	nCurrentPhotonEnergyBitmask : UINT;
	nTargetPhotonEnergyBitmask : UINT;
END_VAR

// Update PVs
fbHgvpuElectronEnergy();

fElectronEnergyVal := fbHgvpuElectronEnergy.fValue;
bElectronEnergyValid := fbHgvpuElectronEnergy.bValid;

fbHgvpu(fbElectronEnergy:=fbHgvpuElectronEnergy);

//Update BP
nCurrentPhotonEnergyBitmask := F_eVRangeCalculator(fbHgvpu.fCurrentPhotonEnergy, nCurrentPhotonEnergyBitmask);
nTargetPhotonEnergyBitmask := F_eVRangeCalculator(fbHgvpu.fTargetPhotonEnergy, nTargetPhotonEnergyBitmask);

BP.neVRange := nCurrentPhotonEnergyBitmask OR nTargetPhotonEnergyBitmask;

END_FUNCTION_BLOCK

// MajorComponents/PMPS_MPS_Interface/FB_BeamClassOutputs
(*
Sets the beam class assertion lines for a given beam class.
*)
FUNCTION_BLOCK FB_BeamClassOutputs
VAR_INPUT
    BP : ST_BeamParams;
END_VAR
VAR_OUTPUT
END_VAR
VAR
    nBeamClass   :    BYTE;
    wBeamClass    :    BYTE;

    InitCounter: BYTE;
    counter    :    INT;
    
    // Beam class lines are restricted to 8 channels in the current design, since
    // there are no plans to use all 16. Channels 1-7 may be allocated to any other
    // beam classes so long as they are ordered least to greatest.
    // Channel 8 is reserved for full beam.
    {attribute 'pytmc' := 'pv: BeamClassChannel
        io: i
        field: DESC Hardwire channel state'}
        epicsBitmap : WORD;
        
    {attribute 'TcLinkTo' := '[1] := TIIB[PMPS_Premp]^Channel 1^Output;
                              [2] := TIIB[PMPS_Premp]^Channel 2^Output;
                              [3] := TIIB[PMPS_Premp]^Channel 3^Output;
                              [4] := TIIB[PMPS_Premp]^Channel 4^Output;
                              
                              [5] := TIIB[PMPS_Premp]^Channel 5^Output;
                              [6] := TIIB[PMPS_Premp]^Channel 6^Output;
                              [7] := TIIB[PMPS_Premp]^Channel 7^Output;
                              [8] := TIIB[PMPS_Premp]^Channel 8^Output;'} // 8 - Full beam
    q_BC_ASSERTION_LINES    AT    %Q*    : ARRAY [1..MAX_BEAM_CLASS_LINES] OF    BOOL;
END_VAR
VAR CONSTANT
    MAX_BEAM_CLASS_LINES : BYTE := 8;
    BC_1HZ : BYTE := 1;
    BC_10HZ : BYTE := 2;
    BC_FULL : BYTE := 16;
END_VAR


// Determine BC
IF BP.nRate >= 120 THEN
    nBeamClass := BC_FULL;
ELSIF BP.nRate >= 10 THEN
    nBeamClass := BC_10HZ;
ELSIF BP.nRate >= 1 THEN
    nBeamClass := BC_1HZ;
ELSE
	nBeamClass := 0;
END_IF


//Assert Beam Class
////////////////////////////////////
//0x0 = 0000 0000 0000 0000
//0x1 = 0000 0000 0000 0001
//0xF = 1111 1111 1111 1111

//Initialize BC lines to zero on every pass
FOR InitCounter := 1 TO MAX_BEAM_CLASS_LINES DO
    q_BC_ASSERTION_LINES[InitCounter] := FALSE;
END_FOR

//Set BC lines according to beam class
//A BC of 0x0 would pass over this loop, setting none of the lines high
// , as FOR loops check the initialized variable at the top to see if it's >
// than the "TO" variable.
FOR wBeamClass:=1 TO MIN(MAX_BEAM_CLASS_LINES-1, nBeamClass) DO
    q_BC_ASSERTION_LINES[wBeamClass] := TRUE;
END_FOR

q_BC_ASSERTION_LINES[8] := nBeamClass = 16; //Set channel 8 true if BC is 16


// Readbacks for EPICS
epicsBitmap.0 := q_BC_ASSERTION_LINES[1];
epicsBitmap.1 := q_BC_ASSERTION_LINES[2];
epicsBitmap.2 := q_BC_ASSERTION_LINES[3];
epicsBitmap.3 := q_BC_ASSERTION_LINES[4];

epicsBitmap.4 := q_BC_ASSERTION_LINES[5];
epicsBitmap.5 := q_BC_ASSERTION_LINES[6];
epicsBitmap.6 := q_BC_ASSERTION_LINES[7];
epicsBitmap.7 := q_BC_ASSERTION_LINES[8];

END_FUNCTION_BLOCK

// MajorComponents/PMPS_MPS_Interface/FB_CTLS_Outputs
(*
Controls auxiliary beam class outputs.

1-3 are mapped to control the Cu beamline rate via the LCLS II MPS.

Maps beam rate requests to 1, 10, or full rate beam for Cu linac.

*)
FUNCTION_BLOCK FB_CTLS_Outputs
VAR_INPUT
    BP    :    ST_BeamParams;
END_VAR
VAR_OUTPUT
END_VAR
VAR
    {attribute 'pytmc' := 'pv: CTLSChannel
        io: i
        field: DESC CTLS Rate Control hardwire channel state'}
    epicsBitmap : WORD;
        
    {attribute 'TcLinkTo' := '[1] := TIIB[PMPS_Premp]^Channel 9^Output;
                              [2] := TIIB[PMPS_Premp]^Channel 10^Output;
                              [3] := TIIB[PMPS_Premp]^Channel 11^Output;'}
    q_CLTS_ASSERTION_LINES    AT    %Q*    : ARRAY [1..3] OF    BOOL;  
    
    
    
END_VAR


// CLTS 1Hz
q_CLTS_ASSERTION_LINES[1] := BP.nRate >= 1;
// CLTS 10Hz
q_CLTS_ASSERTION_LINES[2] := BP.nRate >= 10;
// CLTS Full rate
q_CLTS_ASSERTION_LINES[3] := BP.nRate >= 120;


epicsBitMap.0 := q_CLTS_ASSERTION_LINES[1];
epicsBitMap.1 := q_CLTS_ASSERTION_LINES[2];
epicsBitMap.2 := q_CLTS_ASSERTION_LINES[3];

END_FUNCTION_BLOCK

// MajorComponents/PMPS_MPS_Interface/FB_PhotonEnergyWatcher
(*
A. Wallace 2019-4-22
The photon energy watcher ensures the current and target photon energy is within
the arbirated bounds. Target in this case means, the calculated target photon energy
from the PVs that control the mechatronics of the undulators/ the electron energy.

If there are control PVs that match the monitor PVs, the control PVs are used to 
calculate a "target" photon energy. This is supposed to cover when the undulators/
electron energy is transitioning.

The abritrated bounds come from a simple AND of all the permitted ranges. See
the arbitrate action of the arbiter FB.

Note, this protection logic does not account for beam-off when determining fast-fault
status. If a device is requesting a limited range of eV, this request must be honored,
regardless of current beam-rate.
*)
{attribute 'reflection'}
FUNCTION_BLOCK FB_PhotonEnergyWatcher
VAR_INPUT
    i_stCurrentBeamParams    :    ST_BeamParams; //Link to global beam params
    i_stMachineTargetBeamParams    :    ST_BeamParams; //Link to global machine target beam params
    i_stRequestedBeamParams    :    ST_BeamParams; //Link to arbiter output or beam param. requestor
    // Reset fault
    i_xReset: BOOL;
    sName : STRING := 'PhotonEnergyWatcher';
END_VAR
VAR_OUTPUT
END_VAR
VAR_IN_OUT
    io_fbFFHWO    :    FB_HardwareFFOutput;
END_VAR
VAR
    xPhotonEnergyWithinBounds    :    BOOL;
    fbFF    :    FB_FastFault :=(
        i_DevName := sName,
        i_Desc := 'Fault occurs when the calculated machine photon energy (K value calculated by undulator gap, and electron energy) falls outside the permitted range.',
        i_TypeCode := 7 );
        
   {attribute 'pytmc' := '
        pv: ResidualPhotonEnergies
		io: i
        archive: 1Hz monitor
        field: DESC Portions of beam eV not permitted
        field: EGU eV-bitmask
    '}
    evResidual : WORD;
    
    fbLog : FB_LogMessage := (
        eSubSystem := E_Subsystem.MPS,
        eSevr := TcEventSeverity.Critical
        );
    bLogOneShot : BOOL;
    sDevName : T_MaxString := 'Photon Energy Watcher';
    
    fbGetHN : FB_GetHostName;
    bInit : BOOL := TRUE;
    
    {attribute 'instance-path'}
    {attribute 'noinit'}
    sPath    :    T_MaxString;
    
    fbStr : FB_FormatString := (
        sOut := 'Non-zero photon energy residual: %16b; Req: %16b; Act: %16b');
END_VAR

IF bInit THEN
    fbGetHN(bExecute:=TRUE);
    bInit R= NOT fbGetHN.bBusy;
END_IF
    
xPhotonEnergyWithinBounds := (i_stCurrentBeamParams.neVRange AND i_stRequestedBeamParams.neVRange) = i_stCurrentBeamParams.neVRange;

evResidual := (i_stCurrentBeamParams.neVRange XOR i_stRequestedBeamParams.neVRange) AND i_stCurrentBeamParams.neVRange;

IF evResidual <> 0 AND bLogOneShot THEN
    fbLog.sJson := F_PMPS_JSON(
        CONCAT(fbGetHN.sHostName, sDevName),
        sPath,
        PMPS_CODES.PEW_FAULT);
    
    fbStr.arg1 := F_WORD(evResidual);
    fbStr.arg2 := F_WORD(i_stCurrentBeamParams.neVRange);
    fbStr.arg3 := F_WORD(i_stRequestedBeamParams.neVRange);
    
    fbStr();
        
    fbLog(sMsg:=fbStr.sOut);
    bLogOneShot := FALSE;
ELSIF evResidual = 0 THEN
    bLogOneShot := TRUE;
END_IF

fbFF(i_xOK := xPhotonEnergyWithinBounds,
    io_fbFFHWO := io_fbFFHWO,);

END_FUNCTION_BLOCK

// MajorComponents/SimulationFB/FB_eVSimulator
(* eV Simulator
A. Wallace 2019-8-30

Adds noise to the eV and changes eV position occasionally.
*)
FUNCTION_BLOCK FB_eVSimulator
VAR_INPUT
    NoiseLevel	:	REAL	:= 0; // eV Noise
    ChangeTime : TIME := T#10S;
END_VAR
VAR_OUTPUT
    eV	:	REAL := 300;
END_VAR
VAR
    eVRange : REAL := 1600;
    timer: TON;
    eVRand	:	DRAND :=(Seed:=0);
    NoiseRand : DRAND := (Seed:=0);
END_VAR


timer(in:=TRUE, PT:=ChangeTime);

//Occasionally change eV
IF timer.Q THEN
    timer(in:=FALSE);
    eVRand();
    eV := LIMIT(0, eVRange*LREAL_TO_REAL(eVRand.Num), eVRange);
END_IF

// Noise generation
NoiseRand();
eV := eV + NoiseLevel*LREAL_TO_REAL(NoiseRand.Num);
NoiseRand();
eV := LIMIT(0, ev - NoiseLevel*LREAL_TO_REAL(NoiseRand.Num), eVRange);

END_FUNCTION_BLOCK

// MajorComponents/SimulationFB/FB_MachineSimulator
(* Simulates the machine responding to requests by adding a bit of delay/ ramps
*)
FUNCTION_BLOCK FB_MachineSimulator
VAR_INPUT
    i_stAssertedParams    :    ST_BeamParams;
    i_xFault    :    BOOL;
    
    xEnableAtt : BOOL;
    xEnablePE : BOOL;
    xEnableRate : BOOL;
END_VAR
VAR_IN_OUT
    iq_stMachineParams    :    ST_BeamParams;
END_VAR
VAR
    nTargetTran: UINT;
    tonTranTimer    :    TON := (
        PT := T#2S
        );
    fTargetPP_mJ: REAL;
    tonPPETimer: TON := (
        PT := T#2S
    );
END_VAR


//Attenuation
IF xEnableAtt THEN
    IF i_stAssertedParams.nTran <> nTargetTran THEN
        tonTranTimer(IN:=FALSE);
        nTargetTran := i_stAssertedParams.nTran;
    ELSIF NOT tonTranTimer.Q THEN
        tonTranTimer(IN:=TRUE);
    ELSE
        iq_stMachineParams.nTran := nTargetTran;
    END_IF
END_IF
    
//Pulse Energy
IF xEnablePE THEN
    IF i_stAssertedParams.fPP_mJ <> fTargetPP_mJ THEN
        tonPPETimer(IN:=FALSE);
        fTargetPP_mJ := i_stAssertedParams.fPP_mJ;
    ELSIF NOT tonTranTimer.Q THEN
        tonPPETimer(IN:=TRUE);
    ELSE
        iq_stMachineParams.fPP_mJ := fTargetPP_mJ;
    END_IF
END_IF

//Rate
IF xEnableRate THEN
    IF i_xFault THEN
        iq_stMachineParams.nRate := 0;
    ELSE
        iq_stMachineParams.nRate := i_stAssertedParams.nRate;
    END_IF
END_IF

END_FUNCTION_BLOCK

// MajorComponents/Stoppers/FB_KStopper
FUNCTION_BLOCK FB_KStopper EXTENDS FB_StopperWatcher
VAR_INPUT
END_VAR
VAR_OUTPUT
END_VAR
VAR_IN_OUT
END_VAR
VAR
END_VAR

SUPER^(stCurrentBP:=SUPER^.stCurrentBP);

METHOD FB_init : BOOL
VAR_INPUT
    bInitRetains : BOOL; // if TRUE, the retain variables are initialized (warm start / cold start)
    bInCopyCode : BOOL;  // if TRUE, the instance afterwards gets moved into the copy code (online change)
    eStopper : PMPS.K_Stopper;
    sStopperName : STRING;
END_VAR
Stopper := eStopper;
StopperName := sStopperName;
END_METHOD

END_FUNCTION_BLOCK

// MajorComponents/Stoppers/FB_StopperWatcher
// Relays stopper state and sends a message when stopper state changes.
FUNCTION_BLOCK FB_StopperWatcher
VAR_INPUT
END_VAR
VAR_OUTPUT
END_VAR
VAR_IN_OUT
	stCurrentBP : ST_BeamParams;
END_VAR
VAR
    i_StopperOutLS AT %I* : BOOL;
    i_StopperInLS AT %I* : BOOL;

    q_StopperOUT_Relay AT %Q* : BOOL;
    q_StopperIN_Relay AT %Q* : BOOL;

    Stopper : UINT;
    StopperName : STRING;
	{attribute 'instance-path'}
    {attribute 'noinit'}
    sPath    :    T_MaxString;

    // Logging
    fbLogMsg : FB_LogMessage := (
        eSubSystem := E_Subsystem.MPS);

    rtIn : R_TRIG;
    rtOut : R_TRIG;

	bInit: BOOL := TRUE;
END_VAR

IF bInit THEN
	fbLogMsg.sJson := F_PMPS_JSON(StopperName, sPath, 1000);
	bInit := FALSE;
END_IF


rtIn(CLK := i_StopperInLS);
rtOut(CLK := i_StopperOutLS);

IF rtIn.Q THEN
    fbLogMsg.sMsg := CONCAT(StopperName, ' moved IN');
    fbLogMsg();
ELSIF rtOut.Q THEN
    fbLogMsg.sMsg := CONCAT(StopperName, ' moved OUT');
    fbLogMsg();
END_IF

q_StopperOUT_Relay := i_StopperOutLS;
q_StopperIN_Relay := i_StopperInLS;

// Update current beam parameters
stCurrentBP.aStoppers[Stopper] := i_StopperInLS;

END_FUNCTION_BLOCK

// MajorComponents/Stoppers/FB_LStopper
FUNCTION_BLOCK FB_LStopper EXTENDS FB_StopperWatcher
VAR_INPUT
END_VAR
VAR_OUTPUT
END_VAR
VAR_IN_OUT
END_VAR
VAR
END_VAR

SUPER^(stCurrentBP:=SUPER^.stCurrentBP);

METHOD FB_init : BOOL
VAR_INPUT
    bInitRetains : BOOL; // if TRUE, the retain variables are initialized (warm start / cold start)
    bInCopyCode : BOOL;  // if TRUE, the instance afterwards gets moved into the copy code (online change)
    eStopper : PMPS.L_Stopper;
    sStopperName : STRING;
END_VAR
Stopper := eStopper;
StopperName := sStopperName;
END_METHOD

END_FUNCTION_BLOCK

// MajorComponents/BeamParameterTransitionManager
(*
Implements the procedure for safely transitioning between device states.

NOTE:
The BPTM will throw an error if the arbiter does not have enough space for the transition and new final assertion. 

 *)
FUNCTION_BLOCK BeamParameterTransitionManager
VAR_IN_OUT
    
    fbArbiter    :    FB_Arbiter; //Connect to local arbiter
    
END_VAR
VAR_INPUT
    i_TransitionAssertionID    :    UDINT := 0; // Must not be 0 or EXCLUDED_ID
    i_stTransitionAssertion : ST_BeamParams := PMPS_GVL.cstSafeBeam; //Assertion required during transition (always safer than anything inbetween)
    
    i_nRequestedAssertionID    :    UDINT := 0; // Must not be 0 or EXCLUDED_ID
    i_stRequestedAssertion    :    ST_BeamParams := PMPS_GVL.cstSafeBeam; //Requested assertion, change whenever
    
    i_xMoving    :    BOOL := FALSE; //Provide rising edge when device begins moving <remove>
    i_xDoneMoving    :    BOOL := FALSE; //Provide rising edge when device is done with a move
    
    stCurrentBeamParameters    :    ST_BeamParams := PMPS_GVL.cstFullBeam; //Connect to current beam parameters
    
    // Rising edge to cycle back through the BPTM process. Use if something in the process timed out or failed. This will interrupt a current process
    bRetry : BOOL := FALSE; 
END_VAR
VAR_OUTPUT

    q_xTransitionAuthorized    :    BOOL := FALSE; //Rising edge indicating the device is safe to move, use as input to move execute (which requires a rising edge)

    bError : BOOL; // Set if some issue occurs within the bptm
    nErrId : UINT; // Set to non-zero to help understand the error.
    
    bDone : BOOL;
    bBusy : BOOL;
    
END_VAR

VAR
    nTargetAssertionID    :    UDINT := 0;
    stTargetAssertion    :    ST_BeamParams; // Target assertion
    nCurrentAssertionID    :    UDINT := 0;  // ID of last set state (zero until a state is reached)
    
    xNewBP    :    BOOL;
    xTranBP    :    BOOL;
    xFinalBP    :    BOOL;
    
    eBPTMState : E_BPTMState := Init;
    ePrevState : E_BPTMState := Init;
    
    xEntry : BOOL;
    rTransition : R_TRIG;
    xNewTarget : BOOL;
	
	bTransAssertionFailed : BOOL;
    bFinalAssertionFailed : BOOL;
	
	LogStrBuffer : ARRAY [0..LogBuffSize] OF STRING;
	LogBuffIdx : FB_Index := (LowerLimit:=0, UpperLimit:=LogBuffSize);
    
    nAssrtAttempt : INT; // Number of times we have tried asserting a BP set
    
    rtRetry : R_TRIG;
    
    rtError : R_TRIG;
    
    ffTimeout : FB_FastFault := (
        i_Desc := 'Preemptive requests timed out in BPTM',
        i_TypeCode := 16#A,
        i_xAutoReset := FALSE);
        
	rtDoneMoving : R_TRIG;
    
    bFirstMove : BOOL := TRUE;    
        
END_VAR
VAR CONSTANT
	LogBuffSize : INT := 40;
    cMaxAttempts : INT := 3;
    (* The thought here is, a BPTM needs at most 2 arbiter slots to complete a transition.
    If we're at capacity, it means some BPTM before this one has begun a transition,
    and will require at least one more arbiter spot to complete. 
    *)
    cReqArbCapacity : UDINT := 2;
END_VAR


rtRetry(CLK:=bRetry);
bRetry := FALSE;

rtDoneMoving(CLK:=i_xDoneMoving);

IF nTargetAssertionID <> i_nRequestedAssertionID OR rtRetry.Q THEN
    
    bError := FALSE;
    nErrID := 0;
    
    bDone := FALSE;
    bBusy := TRUE;

    // Execute exit actions before transition back to NewTarget
    CASE eBPTMState OF
        Transitioning:
            DeauthorizeTransition();
        //CleaningUp: 
	END_CASE
        
    eBPTMState := E_BPTMState.NewTarget;
    xEntry := eBPTMState <> ePrevState;
    
END_IF

IF xEntry THEN nAssrtAttempt := 0; END_IF

rtError(CLK:=bError);

IF rtError.Q THEN
    eBPTMState := E_BPTMState.Error;
END_IF

// States
CASE eBPTMState OF
    NewTarget:
        IF xEntry THEN
            NewTarget_ENTRY();
        ELSIF xNewBP THEN
            eBPTMState := E_BPTMState.RequestBP;
        ELSE
            SetNewTarget();
        END_IF
        
    RequestBP:
        IF PMPS_GVL.MAX_ASSERTIONS - fbArbiter.nEntryCount >= cReqArbCapacity THEN
            AssertTransitionBP();
            AssertFinalBP();
            eBPTMState := E_BPTMState.WaitForBP;
		ELSE
            LogActions('Arbiter at capacity, leaving space for other BPTM to finish.');
            nErrId := PMPS_CODES.NoRoomInArb;
            bError := TRUE;
        END_IF
    
    WaitForBP:
        WaitingForTransitionAssertion_DO();
        WaitingForFinalAssertion_DO();
        IF xTranBP AND xFinalBP THEN eBPTMState := E_BPTMState.Transitioning; END_IF
        
    Transitioning:
        IF xEntry THEN
            AuthorizeTransition();
        ELSIF rtDoneMoving.Q OR (bFirstMove AND i_xDoneMoving) THEN
            DeauthorizeTransition();
            eBPTMState := E_BPTMState.CleaningUp;
		END_IF
        
    CleaningUp:
        IF xEntry THEN
            RemoveTransitionAssertion();
		ELSE
			eBPTMState := E_BPTMState.Done;
		END_IF

    Done:
        bDone := TRUE;
        bFirstMove := FALSE;
        LogActions('Returning to idle');
        eBPTMState := E_BPTMState.Idle;
    
    Error:
        bError := TRUE;    
        eBPTMState := E_BPTMState.Idle;
END_CASE

xEntry := ePrevState <> eBPTMState;
ePrevState := eBPTMState;

bDone R= bError;
bBusy R= bError OR bDone;

ACTION AssertFinalBP:
//q_stFinalAssertion := stTargetAssertion;

//Clearing previous target parameters
(* This is considered safe at this step as the transition
state beam parameters should always be safer than the
current or target state beam parameters
*)
IF nCurrentAssertionID <> 0 THEN
    LogActions(CONCAT('Removing previous request: ', DWORD_TO_HEXSTR(nCurrentAssertionID, 4, false)) );
    fbArbiter.RemoveRequest( nCurrentAssertionID );
END_IF

LogActions(CONCAT('Asserting target req.: ', DWORD_TO_HEXSTR(nTargetAssertionID, 4, false)) );

//Asserting target parameters
bFinalAssertionFailed := NOT fbArbiter.AddRequest(
    nTargetAssertionID,
    stTargetAssertion
);

IF bFinalAssertionFailed THEN
    LogActions('Assert final failed. ');
    nAssrtAttempt := nAssrtAttempt + 1;
    IF nAssrtAttempt > cMaxAttempts THEN
        bError := TRUE;
        nErrID := PMPS_CODES.FinalAssrtFail;
    END_IF
ELSE
    // Remembering final assertionID for removal later
    nCurrentAssertionID := nTargetAssertionID;    
END_IF
END_ACTION

ACTION AssertTransitionBP:

LogActions( CONCAT('Removing transition id: ', DWORD_TO_STRING(i_TransitionAssertionID)) );
fbArbiter.RemoveRequest(i_TransitionAssertionID);

LogActions( CONCAT('Requesting transition id: ', DWORD_TO_STRING(i_TransitionAssertionID)) );
bTransAssertionFailed := NOT fbArbiter.AddRequest(
    i_TransitionAssertionID,
    i_stTransitionAssertion
);

IF bTransAssertionFailed THEN
    LogActions('Assert trans. failed. ');
    nAssrtAttempt := nAssrtAttempt + 1;
    IF nAssrtAttempt > cMaxAttempts THEN
        bError := TRUE;
        nErrID := PMPS_CODES.TransAssrtFail;
    END_IF    
END_IF
END_ACTION

ACTION AuthorizeTransition:
q_xTransitionAuthorized := TRUE;

LogActions('Authorizing transition');
END_ACTION

ACTION DeauthorizeTransition:
q_xTransitionAuthorized := FALSE;
LogActions('Deauthorizing transition');
END_ACTION

METHOD LogActions : BOOL
VAR_INPUT
	LogStr : STRING;
END_VAR
LogStrBuffer[LogBuffIdx.IncVal()] := LogStr;
END_METHOD

ACTION NewTarget_ENTRY:
xNewBP := False;
END_ACTION

ACTION RemoveTransitionAssertion:
//q_stTransitionAssertion := PMPS_GVL.cstFullBeam;

//Removing transition assertion
fbArbiter.RemoveRequest( i_TransitionAssertionID );

LogActions('Removing transition req');

//TODO add something to verify removal
END_ACTION

ACTION RequestBP_DO:
// Request BP atomically so we know we'll finish the BPTM cycle
IF fbArbiter.nEntryCount < cReqArbCapacity THEN

    LogActions( CONCAT('Removing transition id: ', DWORD_TO_STRING(i_TransitionAssertionID)) );
    fbArbiter.RemoveRequest(i_TransitionAssertionID);
    
    LogActions( CONCAT('Requesting transition id: ', DWORD_TO_STRING(i_TransitionAssertionID)) );
    bTransAssertionFailed := NOT fbArbiter.AddRequest(
        i_TransitionAssertionID,
        i_stTransitionAssertion
    );
    
    IF bTransAssertionFailed THEN
        LogActions('Assert trans. failed. ');
        nAssrtAttempt := nAssrtAttempt + 1;
        IF nAssrtAttempt > cMaxAttempts THEN
            bError := TRUE;
            nErrID := PMPS_CODES.TransAssrtFail;
        END_IF    
    END_IF
    
    

ELSE
    LogActions('Arbiter at capacity, leaving space for other BPTM to finish.');
END_IF
END_ACTION

ACTION SetNewTarget:

IF F_ValidReqID(i_nRequestedAssertionID) AND
    F_ValidReqID(i_TransitionAssertionID) THEN
    
    stTargetAssertion := i_stRequestedAssertion;
    nTargetAssertionID := i_nRequestedAssertionID;
	
	LogActions('New target set');
	
    xNewBP := TRUE;
    
ELSE
    IF NOT F_ValidReqID(nTargetAssertionID) THEN
        
        nErrID := PMPS_CODES.BadTargetID;
    ELSIF NOT F_ValidReqID(i_TransitionAssertionID) THEN
        nErrID := PMPS_CODES.BadTransID;
	END_IF
    LogActions('Error in set new target');
    bError := TRUE;
END_IF
END_ACTION

ACTION WaitingForFinalAssertion_DO:
//Final Assertion Verification

xFinalBP := F_SafeBPCompare(stCurrentBeamParameters, stTargetAssertion) AND
    fbArbiter.CheckRequest( i_nRequestedAssertionID);;
END_ACTION

ACTION WaitingForFinalAssertion_EXIT:
//Set this bool false so we can get a rising edge on the next try
xFinalBP := FALSE;
END_ACTION

ACTION WaitingForTransitionAssertion_DO:
//Transition Assertion Verification
xTranBP    := F_SafeBPCompare(stCurrentBeamParameters, i_stTransitionAssertion) AND
    fbArbiter.CheckRequest(i_TransitionAssertionID);
END_ACTION

ACTION WaitingForTransitionAssertion_EXIT:
xTranBP := FALSE;
END_ACTION

END_FUNCTION_BLOCK

// MajorComponents/FB_BPControlDevice
(*
Used to request a beam parameter set from EPICS.

Technically just one of these is needed in the entire
PMPS for a line.

*)
FUNCTION_BLOCK FB_BPControlDevice
VAR_INPUT
        (*  Requested pre-optic attenuation %  *)
        {attribute 'pytmc' := 'pv: ReqBP:Transmission
            io: o
            field: EGU %
        '}
        nTran : UINT := 100;
        (* Pulse-rate *)
        {attribute 'pytmc' := 'pv: ReqBP:Rate
            io: o
            field: EGU Hz
        '}
        nRate : UDINT := 10;
        (* Per pulse max energy (mJ) *)
		// non-op
        fPP_mJ : REAL := 20;
        (* Photon energy ranges *)
        {attribute 'pytmc' := 'pv: ReqBP:PhotonEnergyRanges
            io: o
            field: EGU eV'}
        {attribute 'displaymode' := 'binary'}
        neVRange : WORD := 65535;
END_VAR
VAR_OUTPUT
END_VAR
VAR_IN_OUT
    Arbiter : FB_Arbiter;
END_VAR
VAR
    EpicsReqBP : ST_BeamParams;
    {attribute 'pytmc' := '
        pv: ReqBP:Apply
        io: o
    '}
    bApply : BOOL;

    nControlDeviceID : DWORD;

    rtApply : R_TRIG;

END_VAR


EpicsReqBP.nTran := nTran;
EpicsReqBP.neVRange := neVRange;
EpicsReqBP.nRate := nRate;
EpicsReqBP.fPP_mJ := fPP_mJ;

rtApply(CLK:=bApply);
IF rtApply.Q THEN
    Arbiter.RemoveRequest(nControlDeviceID);
    Arbiter.AddRequest(nControlDeviceID, EpicsReqBP);
    bApply := FALSE;
END_IF

METHOD FB_init : BOOL
VAR_INPUT
    bInitRetains : BOOL; // if TRUE, the retain variables are initialized (warm start / cold start)
    bInCopyCode : BOOL;  // if TRUE, the instance afterwards gets moved into the copy code (online change)
    nID : DWORD := PMPS_GVL.EXCLUDED_ASSERTION_ID;
END_VAR
nControlDeviceID:= nID;
END_METHOD

END_FUNCTION_BLOCK

// MajorComponents/FB_BPRequestor
(* BP Requestor
Elevates the BP request from an arbiter to PMPS_GVL.stRequestedBP
*)
FUNCTION_BLOCK FB_BPRequestor IMPLEMENTS I_HigherAuthority
VAR_INPUT
END_VAR
VAR_OUTPUT
    q_ReqBP : ST_BeamParams; // Arbitrated BP
END_VAR
VAR_IN_OUT
    Arbiter : FB_Arbiter;
    //FFO : FB_HardwareFFOutput;
END_VAR
VAR
    ReqBP : ST_BeamParams;
    nCohort : ULINT; // Current cohort, inc. 1 cycle after IO is updated
    nRequestCohort : ULINT; // Cohort number recorded at the time of the request.
END_VAR

Arbiter.ElevateRequest(THIS^); // Executes arbitration and retrieves ReqBP

IF nRequestCohort >= nCohort THEN
    // Update requested BP set
    q_ReqBP := ReqBP;
    // Note: we may do more here someday... perhaps all of the output control
    // will reside in here, and be solely controlled by this block. For now
    // I am going to adopt a flat management structure.
    // Start a new cohort
    nCohort := nCohort + 1;
END_IF

// Returns true when outputs to MPS are updated
METHOD CheckRequest : BOOL
VAR_INPUT
	nReqID	: DWORD;
END_VAR
VAR_INST
    xFirstTime : BOOL;
    nId : DWORD;
END_VAR
(* nRequestCohort will be < nCohort after output control
function blocks have been updated to reflect the new request
*)
CheckRequest := nRequestCohort < nCohort;
END_METHOD

METHOD RemoveRequest : BOOL
VAR_INPUT
	nReqID    :    DWORD; //StateID to remove
END_VAR
END_METHOD

METHOD RequestBP : BOOL
VAR_INPUT
	(*StateID of state requesting beam parameter set*)
	nReqID	: DWORD;
	(*Requested beam params*)
	stReqBP	: ST_BeamParams;
END_VAR
VAR_INST
    ReqID : DWORD;
    Registered : BOOL := FALSE;
END_VAR

// Check the request is coming from the same source we're used to
IF NOT Registered THEN
    ReqID := nReqID;
    Registered := TRUE;
END_IF
// log a complaint if false
RequestBP := ReqId = nReqId;

// Update internal BP request struct
ReqBP := stReqBP;

// Record current cohort

    nRequestCohort := nCohort;
END_METHOD

END_FUNCTION_BLOCK

// MajorComponents/FB_LinearGovernor

(* The governor is meant to check your work and keep you from making mistakes.

Checks:
Does your state match the device position and visa versa?
Are the beam parameters safe for the device state?
Did you properly assert the transition and final beam parameters?

*)
FUNCTION_BLOCK FB_LinearGovernor
VAR_INPUT
    i_stCurrentBeamParams    :    ST_BeamParams; //Link to global beam params
    i_xMPSOverride            :    BOOL; //True releases MPS limits after a delay
    i_xTransitionRequested    :    BOOL; //Set true to request a transition
    i_xResetMPSFault    :    BOOL; //Set true to clear MPS fault 
END_VAR
VAR_OUTPUT
     //True when governor has released restrictions
    q_xTransitionPermitted    :    BOOL;
    //Set if MC_Power has an error, or override mode is requested
    q_xFault    :    BOOL; 
    // Indicates override mode is active
    q_xMPSLimitsOverridden: BOOL;
END_VAR
VAR_IN_OUT
    stDevice    :    ST_Device; //The governed
    Arbiter    :    FB_Arbiter;
    FastFaultOutput    :    FB_HardwareFFOutput;
END_VAR
VAR
    mcPower    :    MC_Power;
    
    xActuatorPositiveEnable: BOOL;
    xActuatorNegativeEnable: BOOL;
    
    xMPSPositiveEnable    :    BOOL;
    xMPSNegativeEnable    :    BOOL;
    lrPosition: LREAL;
    
    lrLatchedTargetPosition    :    LREAL;
    lrLatchedTargetTolerance    :    LREAL;
    stLatchedTargetState    :    ST_DeviceStateExt;
    
    lrMPSUpperLimit: LREAL;
    lrMPSLowerLimit: LREAL;
    rtNewState: R_TRIG;
    xTransitionOK: BOOL;
    
    tonMPSOverrideMode    :    TON := (
        PT := T#5S
    );
    
    srMPSFault    :    SR;
    // Actuator out of bounds fault
    xActuatorOOB: BOOL;
    //Beam parameters out of spec
    xBeamParamsOOS: BOOL;
    //Beam parameters of currently latched state
    
    stLatchedBeamParams: ST_BeamParams;
    stTargetState: ST_DeviceStateExt;
    
    rtLatchNewState    :    R_TRIG;
    xInit: BOOL := TRUE;
    
    stInitDeviceState: ST_DeviceStateExt;
    // Indicates an error with initialization
    xInitFault: BOOL;
    // Indicates the state could not be found in the state table. There may be something wrong in the device state machine implementation or state table instantiation.
    xStateLookupError: BOOL;
    // A transition needs to be requested at least once before we start latching any state.
    xTransitionHasBeenRequested: BOOL := FALSE;
    ffBeamParamsOK : FB_FastFault;
    ffActuatorBoundsOK    :    FB_FastFault;
END_VAR


lrPosition := stDevice.stAxis.NcToPlc.ActPos; //Actuator position

stDevice.stAxis.ReadStatus();
//Init
(* The init strategy is:
If the device is restored and it's residing at the safe position,
no PMPS faults. *)
////////////////////////////////
    IF xInit THEN
        xInit := FALSE;
        //Use nSafeSate for initialization. 
        stDevice.StateTable.A_Lookup(key := stDevice.nSafeState);
        IF stDevice.StateTable.bOk THEN
            stInitDeviceState := F_DeviceState_To_DeviceStateExt(stDevice.StateTable.getValue, TRUE);
            xInitFault := FALSE;
        ELSE
            xInitFault := TRUE;
            stInitDeviceState.xValid := FALSE;
        END_IF
        lrLatchedTargetPosition := stInitDeviceState.rPosition;
        lrLatchedTargetTolerance := stInitDeviceState.rTolerance;
        stLatchedBeamParams := stInitDeviceState.stReqBeamParam;
    END_IF

// The governor will permit transitions once it verifies the transition assertion is active
// Note the governor does not verify the target state beam params are asserted, perhaps it should <TODO>
////////////////////////////////
    IF i_xTransitionRequested THEN
        xTransitionHasBeenRequested    := TRUE;
        
        xTransitionOK := Arbiter.CheckRequest( stDevice.stTransitionState.nStateRef) AND F_SafeBPCompare(i_stCurrentBeamParams, stDevice.stTransitionState.stReqBeamParam);
        
        //Set the target state for evaluation in further logic
        stdevice.StateTable.A_Lookup(key := stDevice.nTargetState);
        IF stDevice.StateTable.bOk THEN
            stTargetState := F_DeviceState_To_DeviceStateExt(stDevice.StateTable.getValue, TRUE);
            xStateLookupError := FALSE;
        ELSE
            xStateLookupError := TRUE;
            stTargetState.xValid := FALSE;
        END_IF
    ELSE
        xTransitionOK := FALSE;
    END_IF

(* Note about TransitionRequested

If TransitionRequested goes false during a transition, an MPS fault may be induced. This occurs
because the Actuator Out of Bounds fault will go back to using the original state limits, which
the axis may have already moved beyond.

To avoid this transient fault, make sure your device state machine is implemented such that the 
transition request to the governor block remains high until the target position is reached.
*)

//Determine if a transition is complete and latch the new state
(* A transition is complete when:

Axis at standstill.
Axis within tolerance.
No transition req.

Once these conditions are met, the MPS limits shall re-engage to restrict the
axis motion to the tolerance around the state position and the MPS fault monitors
shall evaluate based on the newly latched target state.
*)

rtLatchNewState(CLK := stDevice.stAxis.Status.StandStill AND
    lrPosition <= stTargetState.rPosition + stTargetState.rTolerance AND
    lrPosition >= stTargetState.rPosition - stTargetState.rTolerance AND
    NOT i_xTransitionRequested AND xTransitionHasBeenRequested);
    
IF rtLatchNewState.Q THEN
    lrLatchedTargetPosition := stTargetState.rPosition;
    lrLatchedTargetTolerance := stTargetState.rTolerance;
    stLatchedBeamParams := stTargetState.stReqBeamParam;
    stLatchedTargetState := stTargetState;
END_IF

//Let other blocks know the governor won't interfer with transitions
q_xTransitionPermitted := xTransitionOK;

//Adjust limit ranges based on active state and current target
IF xTransitionOK THEN
    //Extend range to include target state
    lrMPSUpperLimit := MAX(lrMPSUpperLimit, stTargetState.rPosition + stTargetState.rTolerance);
    lrMPSLowerLimit := MIN(lrMPSLowerLimit, stTargetState.rPosition - stTargetState.rTolerance);
ELSE
    //Calculate the limit positions for MPS based on current state
    lrMPSUpperLimit := lrLatchedTargetPosition + lrLatchedTargetTolerance;
    lrMPSLowerLimit := lrLatchedTargetPosition - lrLatchedTargetTolerance;
END_IF


//MPS override
(* In override mode, the device will be free to move anywhere within it's travel range *)
//Permit motion after a small delay
tonMPSOverrideMode(IN:=i_xMPSOverride OR stDevice.xOverrideMPSLimits, Q=>q_xMPSLimitsOverridden);

//Virtual limit switch evaluation
xActuatorPositiveEnable    := stDevice.i_xHiLim AND lrPosition <= stDevice.lrUpperPositionLimit;
xActuatorNegativeEnable    := stDevice.i_xLoLim AND lrPosition >= stDevice.lrLowerPositionLimit;

//Evaluate MPS limit states
xMPSPositiveEnable := lrPosition <= lrMPSUpperLimit;
xMPSNegativeEnable := lrPosition >= lrMPSLowerLimit;

//Final Limit switch evaluation
mcPower.Enable_Positive := xActuatorPositiveEnable AND (tonMPSOverrideMode.Q OR xMPSPositiveEnable);
mcPower.Enable_Negative := xActuatorNegativeEnable AND (tonMPSOverrideMode.Q OR xMPSNegativeEnable);

mcPower(
    Axis := stDevice.stAxis,
    Enable := stDevice.xEnable //link to device enable <TODO>
);



//MPS Faults
//Fault if the beam is unsafe for current state
ffBeamParamsOK(i_xOK:=F_SafeBPCompare(i_stCurrentBeamParams, stLatchedBeamParams), 
                i_xReset:=i_xResetMPSFault,
                io_fbFFHWO := FastFaultOutput);

//Fault if the position is outside of the permitted range
ffActuatorBoundsOK(i_xOK := (lrPosition <= lrMPSUpperLimit AND lrPosition >= lrMPSLowerLimit), 
                    i_xReset:=i_xResetMPSFault,
                io_fbFFHWO := FastFaultOutput);


    
//Collect all other faults
q_xFault := NOT ffBeamParamsOK.o_xFFLine OR
    NOT ffActuatorBoundsOK.o_xFFLine OR
    mcPower.Error    OR
    i_xMPSOverride    OR
    xInitFault;

//Any faults trip the fast fault line for this FB    
//FastFaultOutput.CheckIn(NOT q_xFault);

END_FUNCTION_BLOCK

// MajorComponents/FB_LRateFromEPICS
FUNCTION_BLOCK FB_LRateFromEPICS

(*
enum MPSBeamRates {
    MPSRateInvalid            =  0,
    MPSRate0Hz                =  1,
    /* Previously used 2 and 3 for single shot and burst */
    MPSRate1Hz                =  4,
    MPSRate10Hz               =  5,
    MPSRate30Hz               =  6,
    MPSRate60Hz               =  7,
    MPSRate120Hz              =  8,
    MPSRateUnknown            =  9,
    MPSRateSingleShot         = 10,
    MPSRateBurstMode          = 11,
    MPSRateBurstModeNotActive = 12,
    MPSNumberOfBeamRates      = 13,
    MPSRateBurstInvalid       = 14
}
*)

VAR_IN_OUT
	BP : ST_BeamParams;
END_VAR
VAR_OUTPUT
	xError : BOOL;
END_VAR
VAR
	{attribute 'pytmc' := '
        pv: L:Rate
        link: IOC:BSY0:MP01:BYKIK_RATE
        field: EGU RateEnum
    '}
    fbBYKIK_Rate : FB_LREALFromEPICS;
	
	eMPSRate : E_MPSBeamRates;
END_VAR
VAR CONSTANT
	cFailSafeRate : UINT := 120;
END_VAR

fbBYKIK_Rate();

eMPSRate := LREAL_TO_UINT(fbBYKIK_Rate.fValue);

CASE eMPSRate OF
	MPSRateInvalid:
		BP.nRate := cFailSafeRate;
	MPSRate0Hz:
		BP.nRate := 0;
	MPSRate1Hz:
		BP.nRate := 1;
	MPSRate10Hz:
		BP.nRate := 10;
	MPSRate30Hz:
		BP.nRate := 30;
	MPSRate60Hz:
		BP.nRate := 60;
	MPSRate120Hz:
		BP.nRate := 120;
	MPSRateUnknown:
		BP.nRate := cFailSafeRate;
	
ELSE
	BP.nRate := cFailSafeRate;
END_CASE

BP.xValid R= NOT fbBYKIK_Rate.bValid OR
			eMPSRate = MPSRateUnknown OR
			eMPSRate = MPSRateInvalid;

END_FUNCTION_BLOCK

// MajorComponents/FB_RateFromEPICS
FUNCTION_BLOCK FB_RateFromEPICS

(*
enum MPSBeamRates {
    MPSRateInvalid            =  0,
    MPSRate0Hz                =  1,
    /* Previously used 2 and 3 for single shot and burst */
    MPSRate1Hz                =  4,
    MPSRate10Hz               =  5,
    MPSRate30Hz               =  6,
    MPSRate60Hz               =  7,
    MPSRate120Hz              =  8,
    MPSRateUnknown            =  9,
    MPSRateSingleShot         = 10,
    MPSRateBurstMode          = 11,
    MPSRateBurstModeNotActive = 12,
    MPSNumberOfBeamRates      = 13,
    MPSRateBurstInvalid       = 14
}
*)

VAR_IN_OUT
	BP : ST_BeamParams;
    fbBYKIK_Rate : FB_LREALFromEPICS;
END_VAR
VAR_OUTPUT
	xError : BOOL;
END_VAR
VAR

	
	eMPSRate : E_MPSBeamRates;
END_VAR
VAR CONSTANT
	cFailSafeRate : UINT := 120;
END_VAR

fbBYKIK_Rate();

eMPSRate := LREAL_TO_UINT(fbBYKIK_Rate.fValue);

CASE eMPSRate OF
	MPSRateInvalid:
		BP.nRate := cFailSafeRate;
	MPSRate0Hz:
		BP.nRate := 0;
	MPSRate1Hz:
		BP.nRate := 1;
	MPSRate10Hz:
		BP.nRate := 10;
	MPSRate30Hz:
		BP.nRate := 30;
	MPSRate60Hz:
		BP.nRate := 60;
	MPSRate120Hz:
		BP.nRate := 120;
	MPSRateUnknown:
		BP.nRate := cFailSafeRate;
	
ELSE
	BP.nRate := cFailSafeRate;
END_CASE

BP.xValid R= NOT fbBYKIK_Rate.bValid OR
			eMPSRate = MPSRateUnknown OR
			eMPSRate = MPSRateInvalid;

END_FUNCTION_BLOCK

// TestComponents/FB_Arbiter_Test
{attribute 'call_after_init'}
FUNCTION_BLOCK FB_Arbiter_Test EXTENDS TcUnit.FB_TestSuite
VAR_INPUT
END_VAR
VAR_OUTPUT
END_VAR
VAR
END_VAR

Arbitration();
RequestCheckRemoveBP();
FullArbitrationStack();
StackArbiters();

METHOD ArbiterCapacity
VAR_INPUT
END_VAR
VAR   
    nId    :    DWORD := 1;
    stReq    :    ST_BeamParams := (nTran:=12);
    
    nRandID : DWORD;
    testReq : ST_BeamParams := (neVRange := 16#FFEE, nRate:=33);
    
    idx : DWORD;

END_VAR
VAR_INST
    fbArbCapacityTest    :    FB_Arbiter(1);

    Cycle : INT := 0;
    
    CycleLimit : INT := 20;
    
END_VAR
VAR CONSTANT
    SysID : DWORD := 42;
END_VAR

TEST('Arbiter Capcity');
    // Fill the arbiter
    FOR idx := 1 TO PMPS_GVL.MAX_ASSERTIONS DO
        fbArbCapacityTest.AddRequest(nReqID := idx, stReqBP := testReq);
    END_FOR

TEST_FINISHED();
END_METHOD

METHOD Arbitration
VAR_INPUT
END_VAR
VAR
    
     nTranReqID    :    UDINT    := 1;
    stAttReqBP    :    ST_BeamParams := PMPS_GVL.cstFullBeam;
    
    nPPEReqID    :    UDINT    := 2;
    stPPEReqBP    :    ST_BeamParams := PMPS_GVL.cstFullBeam;
    
    nEVReqID    :    UDINT    := 3;
    stEVReqBP    :    ST_BeamParams := PMPS_GVL.cstFullBeam;
    
    nRateReqID    :    UDINT    := 4;
    stRateReqBP    :    ST_BeamParams := PMPS_GVL.cstFullBeam;
    
    stArbitratedBP    :    ST_BeamParams;
    stExpectedBP    :    ST_BeamParams;
END_VAR
VAR_INST
    fbArbiter    :    FB_Arbiter(1);
END_VAR
TEST('Arbitration');

stAttReqBP.nTran := 50;
stPPEReqBP.fPP_mJ := 1;
stEVReqBP.neVRange := 2#1111_1100_1111_1111;
stRateReqBP.nRate := 10;

stExpectedBP.nTran     :=     stAttReqBP.nTran;
stExpectedBP.fPP_mJ    :=  stPPEReqBP.fPP_mJ;
stExpectedBP.neVRange := stEVReqBP.neVRange;
stExpectedBP.nRate := stRateReqBP.nRate;

//Load arbiter with beam parameter sets
AssertTrue(fbArbiter.AddRequest(nTranReqID, stAttReqBP),
                    'Safest attenuation request failed to load');
                    
//Load arbiter with beam parameter sets
AssertTrue(fbArbiter.AddRequest(nPPEReqID, stPPEReqBP),
                    'Safest PPE request failed to load');
                    
//Load arbiter with beam parameter sets
AssertTrue(fbArbiter.AddRequest(nEVReqID, stEVReqBP),
                    'Safest stEVReqBP request failed to load');
                    
//Load arbiter with beam parameter sets
AssertTrue(fbArbiter.AddRequest(nRateReqID, stRateReqBP),
                    'Safest stRateReqBP request failed to load');

stArbitratedBP := fbArbiter.GetArbitratedBP();

AssertFalse(F_DifferentBeamParams(stExpectedBP, stArbitratedBP),
                'Arbitrated BP does not match expected.');

TEST_FINISHED();
END_METHOD

METHOD FullArbitrationStack
VAR_INPUT
END_VAR
VAR   
    nId    :    DWORD := 1;
    stReq    :    ST_BeamParams := (nTran:=12);
	
	nIdDoS : DWORD := 13;
	stDoSReq : ST_BeamParams := PMPS_GVL.cstFullBeam;
END_VAR
VAR_INST
    fbArbiter    :    FB_Arbiter(1);
    
    fbHigherArb : FB_Arbiter(2);
    
    fbSubSysToArb : FB_SubSysToArbiter_IO; // Subsystem interface with beamline arbiter PLC
    pBPR : POINTER TO ST_BeamParams_IO;
    
    fbArbToSubSys : FB_ArbiterToSubSys_IO := (RequestingSystemID:=42); // Beamline arbiter PLC interface with subsystems
    pBPC : POINTER TO ST_BeamParams_IO;
    
    fbBPR : FB_BPRequestor; // Use in the arbiter PLC to apply an arbitrated beam parameter set to the accelerator interface
    
    FFO : FB_HardwareFFOutput; // Dummy FFO not important for these tests

    Cycle : INT := 0;
    
    CycleLimit : INT := 20;
    
END_VAR
VAR CONSTANT
    SysID : DWORD := 42;
END_VAR
// This simulates a synchronous cycle between the subsystem and arbiter PLC cycles. Ie. phase is locked, and cycle time is the same. This is not always the case, so these tests should be 
// trusted with a grain of salt.

TEST('FullStack');



CASE Cycle OF

0: 
    IF NOT fbArbiter.CheckRequestInPool(nID) THEN
        AssertTrue(fbArbiter.AddRequest(nId, stReq), 'Arbiter returned false from AddRequest'); // some device asking its local arbiter for some beam parameters
    END_IF  
    
    TEST('JustEnteredRequest');
    AssertFalse(fbArbiter.CheckRequest(nId),
        'Check should fail. Request not arbitrated yet.');
    TEST_FINISHED();
   
8000:
    TEST_FINISHED_NAMED('FullStack');   
    
END_CASE 


TEST('VerifyBPRHasBP');
IF fbHigherArb.CheckRequest(SysID) THEN
    AssertFalse(F_DifferentBeamParams(stReq, fbBPR.q_ReqBP),
        'Beam parameters not fully propagated to BPR at highest level');
        TEST_FINISHED_NAMED('VerifyBPRHasBP');
END_IF

TEST('ArbToSubsysPropagation');
IF fbArbToSubSys.nActiveCohort = fbArbToSubSys.nRequestedCohort 
    AND fbArbToSubSys.nActiveCohort <> 0 THEN
    AssertTrue(fbHigherArb.CheckRequest(SysID),
        'Active cohort = Requested cohort before higher arbiter confirmed request was active');
    TEST_FINISHED_NAMED('ArbToSubsysPropagation');
END_IF

TEST('SubsysToArbPropagation');
IF fbArbiter.CheckRequest(nId) THEN
    AssertTrue(fbSubSysToArb.nActiveCohort >= fbSubSysToArb.nRequestCohort,
        'Request validated before higher level confirmation');
    TEST_FINISHED_NAMED('SubsysToArbPropagation');
END_IF


TEST('VerifyIncludedAtAllLevels');
IF fbArbiter.CheckRequest(nId) THEN
    AssertTrue(fbHigherArb.xActiveInArbitration, 'HigherArb is not yet included in arbitration');
    AssertTrue(fbArbiter.xActiveInArbitration, 'Local Arb is not yet included in arbitration');
    TEST_FINISHED_NAMED('VerifyIncludedAtAllLevels');
END_IF
      
    
///////////////////////////////////////
//Sub system cycle
fbSubSysToArb(Arbiter := fbArbiter, fbFFHWO := FFO);
//END of sub system cycle
///////////////////////////////////////

//Ethercat transfer simulation
// Transfer of requested BP to arbiter PLC
pBPR := ADR(fbArbToSubSys.i_RequestedBP);
pBPR^ := fbSubSysToArb.q_stRequestedBP;

// Transfer of current BP to sub system PLC
pBPC := ADR(fbSubSysToArb.i_stCurrentBP);
pBPC^ := fbArbToSubSys.o_CurrentBP;

//////////////////////////////////////
//Start of arbiter plc cycle
//Arb io collects sub system status
fbArbToSubSys(Arbiter := fbHigherArb, fbFFHWO := FFO); // This is making a request in the higher arb
//BPR collects arbiter summation
fbBPR(Arbiter := fbHigherArb); // This is getting the arbitrated BP




IF CycleLimit > Cycle THEN
    Cycle := Cycle + 1;
ELSE 
    Cycle := 8000;
END_IF
END_METHOD

METHOD RequestCheckRemoveBP
VAR_INPUT
END_VAR
VAR
    
    nId    :    DWORD := 1;
    stReq    :    ST_BeamParams;
END_VAR
VAR_INST
    fbArbiter    :    FB_Arbiter(1);
END_VAR
TEST('RequestBP');
AssertTrue(fbArbiter.AddRequest(nId, stReq),
    'Request failed');

TEST_FINISHED();
    
TEST('DuplicateID');
AssertFalse(fbArbiter.AddRequest(nId, stReq),
    'Duplicate request accepted, not good.');

TEST_FINISHED();
    
TEST('CheckBP');
AssertFalse(fbArbiter.CheckRequest(nId),
    'Check should fail. Request not arbitrated yet.');
TEST_FINISHED();

TEST('CheckBPArbitrated');
WRITE_PROTECTED_ULINT(ADR(fbArbiter.nArbiterCohort), fbArbiter.nArbiterCohort + 1);
WRITE_PROTECTED_BOOL(ADR(fbArbiter.xActiveInArbitration), TRUE);
AssertTrue(fbArbiter.CheckRequest(nId),
    'Check should pass.');

TEST_FINISHED();      
    
TEST('IDDoesNotExist');
WRITE_PROTECTED_ULINT(ADR(fbArbiter.nArbiterCohort), fbArbiter.nArbiterCohort + 1); 
AssertFalse(fbArbiter.CheckRequest(nId+1),
    'Check returned true when ID does not exist');

TEST_FINISHED();
    
TEST('RemoveBP');
AssertTrue(fbArbiter.RemoveRequest(nId),
    'Remove failed');
AssertFalse(fbArbiter.CheckRequest(nId),
    'Remove did not remove request');
    
TEST_FINISHED();

TEST('NoRequestsFullBeam');

AssertFalse(F_DifferentBeamParams(fbArbiter.GetArbitratedBP(), PMPS_GVL.cstFullBeam), 'Arbitrated beam should be full with all requests removed');

TEST_FINISHED();
END_METHOD

METHOD StackArbiters
VAR_INPUT
END_VAR
VAR   
    nId    :    DWORD := 1;
    stReq    :    ST_BeamParams := (nTran:=12);
END_VAR
VAR_INST
    fbArbiter    :    FB_Arbiter(1);
    
    fbHigherArb : FB_Arbiter(2);
	
	ArbBP : ST_BeamParams;

    Cycle : INT := 0;
    
    CycleLimit : INT := 20;
    
END_VAR
VAR CONSTANT
    SysID : DWORD := 42;
END_VAR

TEST('StackingArbiters');
fbArbiter.AddRequest(nReqID:=nId, stReqBP:=stReq);

fbArbiter.ElevateRequest(fbHigherArb);

ArbBP := fbHigherArb.GetArbitratedBP();

AssertTrue(ArbBP.nTran = 12, 'We should see the transmission number here');

TEST_FINISHED();
END_METHOD

END_FUNCTION_BLOCK

// TestComponents/FB_ArbToSubsys_Test
{attribute 'call_after_init'}
FUNCTION_BLOCK FB_ArbToSubsys_Test EXTENDS TcUnit.FB_TestSuite
VAR_INPUT
END_VAR
VAR_OUTPUT
END_VAR
VAR
END_VAR

BasicFunction();

METHOD BasicFunction
VAR_INPUT
END_VAR
VAR CONSTANT
    SysID : DWORD := 42;
END_VAR
VAR   
    nId    :    DWORD := 1;
    stReq    :    ST_BeamParams := (nTran:=12);
END_VAR
VAR_INST
    fbArbiter    :    FB_Arbiter(1);
    
    pBPR : POINTER TO ST_BeamParams_IO;
    
    stBPRIO : ST_BeamParams_IO := (
        nCohortInt := 1,
        nTran := 35); // Simulates subsystem BP request
    
    fbArbToSubSys : FB_ArbiterToSubSys_IO := (RequestingSystemID:=42); // Beamline arbiter PLC interface with subsystems
    pBPC : POINTER TO ST_BeamParams_IO;
    
    fbBPR : FB_BPRequestor; // Use in the arbiter PLC to apply an arbitrated beam parameter set to the accelerator interface
    
    FFO : FB_HardwareFFOutput; // Dummy FFO not important for these tests

    Cycle : INT := 0;
    
    CycleLimit : INT := 20;
    
END_VAR

// Simulate an initial cycle with no new requests coming in
fbBPR(Arbiter:=fbArbiter);
fbArbToSubSys(Arbiter:=fbArbiter, fbFFHWO:=FFO);

TEST('Init');
TEST_FINISHED();

//Ethercat transfer simulation
// Transfer of requested BP to arbiter PLC
pBPR := ADR(fbArbToSubSys.i_RequestedBP);
pBPR^ := stBPRIO;

///////////////////////////////////////
//Sub system cycle
fbBPR(Arbiter:=fbArbiter);
fbArbToSubSys(Arbiter:=fbArbiter, fbFFHWO:=FFO);
//END of sub system cycle
///////////////////////////////////////


TEST('New request');
    AssertTrue(fbArbToSubSys.nRequestedCohort = fbArbToSubSys.i_RequestedBP.nCohortInt, 'ReqCohort and qBP Cohort do not match, and they should');
    AssertTrue(fbArbiter.CheckRequestInPool(SysID), 'ArbToSubSys request should be in arbiter pool now');
    AssertTrue(fbArbToSubSys.nActiveCohort = 0, 'Active cohort should remain the initial value until the current request is active in higher arbitration');
    AssertTrue(fbArbToSubSys.o_CurrentBP.nCohortInt = fbArbToSubSys.nActiveCohort, 'Cohort being sent to sub system remains unincremented');
TEST_FINISHED_NAMED('New request');
    

///////////////////////////////////////
//Sub system cycle
fbBPR(Arbiter:=fbArbiter);
fbArbToSubSys(Arbiter:=fbArbiter, fbFFHWO:=FFO);
//END of sub system cycle
///////////////////////////////////////

///////////////////////////////////////
//Sub system cycle
fbBPR(Arbiter:=fbArbiter);
fbArbToSubSys(Arbiter:=fbArbiter, fbFFHWO:=FFO);
//END of sub system cycle
///////////////////////////////////////

///////////////////////////////////////
//Sub system cycle
fbBPR(Arbiter:=fbArbiter);
fbArbToSubSys(Arbiter:=fbArbiter, fbFFHWO:=FFO);
//END of sub system cycle
///////////////////////////////////////

TEST('Request has become active');
    AssertTrue(fbArbToSubSys.nRequestedCohort = fbArbToSubSys.nActiveCohort, 'ReqCohort and qBP Cohort do not match, and they should');
    AssertTrue(fbArbiter.CheckRequest(SysID), 'ArbToSubSys request should be in arbiter pool now');
    AssertTrue(fbArbToSubSys.nActiveCohort = stBPRIO.nCohortInt, 'Active cohort should remain the initial value until the current request is active in higher arbitration');
    AssertTrue(fbBPR.q_ReqBP.nTran = stBPRIO.nTran, 'BPR and requested BP should match');
TEST_FINISHED_NAMED('Request has become active');
END_METHOD

END_FUNCTION_BLOCK

// TestComponents/FB_AttenuatorSimulator
FUNCTION_BLOCK FB_AttenuatorSimulator
VAR_INPUT
    i_rRequestedAttenuation    :    REAL;
    i_stBPReadback    :    ST_BeamParams;
END_VAR
VAR_OUTPUT
    q_xFault    :    BOOL;
    q_rCurrentAttenuation    :    REAL;
END_VAR
VAR_IN_OUT
    Arbiter    :    FB_Arbiter; //Higher level arbiter from which upstream attenuation can be requested
END_VAR
VAR
    tonDelay    :    TON := (
        PT := T#3S
        );
END_VAR

// Really basic delay
tonDelay(IN := i_rRequestedAttenuation <> q_rCurrentAttenuation);

IF tonDelay.Q THEN
    q_rCurrentAttenuation := i_rRequestedAttenuation;
END_IF

END_FUNCTION_BLOCK

// TestComponents/FB_BPTM_Test
{attribute 'call_after_init'}
FUNCTION_BLOCK FB_BPTM_Test EXTENDS TcUnit.FB_TestSuite
VAR_INPUT
END_VAR
VAR_OUTPUT
END_VAR
VAR
END_VAR
VAR CONSTANT
    BPTM_ARR : UDINT := PMPS_GVL.MAX_ASSERTIONS;
END_VAR

BPTMBasicFunction();
//InterruptedTransition();
FullArbError();

METHOD BPTMBasicFunction
VAR_INPUT
END_VAR
VAR    
    //Final and transition assertions
    nTransitionID    :    UDINT := 1;
    stTransitionAssertion    :    ST_BeamParams := (nRate := 10);
    
    nReqID    :    UDINT    := 2;
    stReqAssertion    :    ST_BeamParams := (nTran := 20);
    
END_VAR
VAR_INST
    fbBPTM_TestBasicFunction    :    BeamParameterTransitionManager;
    fbArbiter    :    FB_Arbiter(1);
    ffo : FB_HardwareFFOutput;
    fbSubSysIO : FB_DummyArbIO;
    xFirstPass    :    BOOL := TRUE;
    eTestStep: E_BPTMTestStates := E_BPTMTestStates.Init;
END_VAR

// Completes arbiter request elevation process
// Necessary for CheckRequest to return true, ever
    fbBPTM_TestBasicFunction(
        fbArbiter := fbArbiter,
        stCurrentBeamParameters := fbSubSysIO.q_stSimulatedBPReadback);

fbSubSysIO(LA := fbArbiter, FFO := ffo);

CASE eTestStep OF

E_BPTMTestStates.Init:
    
    TEST('BPTMTest');
    eTestStep := E_BPTMTestStates.WaitingForBeam;

E_BPTMTestStates.WaitingForBeam:
    TEST('BPTM Waits for Beam');
    
    fbBPTM_TestBasicFunction.i_TransitionAssertionID := nTransitionID;
    fbBPTM_TestBasicFunction.i_stTransitionAssertion := stTransitionAssertion;
    
    fbBPTM_TestBasicFunction.i_nRequestedAssertionID := nReqID;
    fbBPTM_TestBasicFunction.i_stRequestedAssertion := stReqAssertion;
    
    IF fbBPTM_TestBasicFunction.eBPTMState = E_BPTMState.WaitForBP AND 
        NOT fbBPTM_TestBasicFunction.xEntry THEN
    
        AssertTrue(fbArbiter.CheckRequestInPool(nTransitionID), 'Arbiter did not accept BPTM transition assertion');
        
        AssertTrue(fbArbiter.CheckRequestInPool(nReqID), 'Arbiter did not accept BPTM transition assertion');
                
        AssertFalse(fbBPTM_TestBasicFunction.q_xTransitionAuthorized,
            'Transition should not be authorized until requests are in and beam is ready');
            
        AssertTrue(fbBPTM_TestBasicFunction.bBusy, 'Busy should be true here');
        AssertFalse(fbBPTM_TestBasicFunction.bDone, 'Done should be false');
        AssertFalse(fbBPTM_TestBasicFunction.bError, 'Error should be false here');
            
        TEST_FINISHED_NAMED('BPTM Waits for Beam');
        
        eTestStep := E_BPTMTestStates.Transitioning;
    END_IF


E_BPTMTestStates.Transitioning:
    TEST('BPTM Authorizes Transition');

    fbSubSysIO.ApplyBPReq(TRUE);    
    
    IF fbBPTM_TestBasicFunction.eBPTMState = E_BPTMState.Transitioning AND
        NOT fbBPTM_TestBasicFunction.xEntry THEN
    
        AssertTrue(fbArbiter.CheckRequest(nReqID),
            'Transition assertion should be in arbiter');
        
        AssertTrue(fbArbiter.CheckRequest(nReqID),
            'Final assertion should be in arbiter');
            
        AssertTrue(fbBPTM_TestBasicFunction.q_xTransitionAuthorized,
            'Transition should be authorized at this point.');
            
        AssertEquals(nReqID, fbBPTM_TestBasicFunction.nCurrentAssertionID,
            'nCurrentAssertionID not set.');
    
        TEST_FINISHED_NAMED('BPTM Authorizes Transition');
        
        eTestStep := E_BPTMTestStates.CleaningUp;
    END_IF

E_BPTMTestStates.CleaningUp:

    TEST('Cleaning up');
    
    fbBPTM_TestBasicFunction.i_xDoneMoving := TRUE;
    
    IF fbBPTM_TestBasicFunction.eBPTMState = E_BPTMState.Done THEN
        
        AssertFalse(fbArbiter.CheckRequestInPool(nTransitionID), 'Transition req should be removed from arb now');
        
        eTestStep := E_BPTMTestStates.Done; 
        
        TEST_FINISHED_NAMED('Cleaning up');
	END_IF

E_BPTMTestStates.Done:

    
    AssertTrue(fbBPTM_TestBasicFunction.bDone, 'Done should be set');
    AssertFalse(fbBPTM_TestBasicFunction.bError, 'Error should be cleared');
    AssertFalse(fbBPTM_TestBasicFunction.bBusy, 'Busy should be false');
    
    TEST_FINISHED_NAMED('BPTMTest');    
    
END_CASE
END_METHOD

// Simulate error due to full arbiter
METHOD FullArbError
VAR_INPUT
END_VAR
VAR    
    //Final and transition assertions
    nTransitionID    :    UDINT := 1000;
    stTransitionAssertion    :    ST_BeamParams := PMPS_GVL.cstSafeBeam;
    
    nReqID    :    UDINT    := 2000;
    stReqAssertion    :    ST_BeamParams := PMPS_GVL.cstSafeBeam;
    
    idx : UDINT;
    
    nRandID : DWORD;
    testReq : ST_BeamParams := (neVRange := 16#FFEE, nRate:=33);
    
END_VAR
VAR_INST
    fbBPTM_TestFullArb    :    BeamParameterTransitionManager;
    fbArbFullErr    :    FB_Arbiter(1);
    ffo : FB_HardwareFFOutput;
    fbSubSysIO : FB_DummyArbIO;
    fbBPR :  FB_BPRequestor;
    xFirstPass    :    BOOL := TRUE;
    eTestStep: E_BPTMTestStates := E_BPTMTestStates.Init;
    tonRetryTimeout : TON := (PT:=T#5s);
    entryToRetry : bool := true;
    fbRand : DRAND := (Seed :=1);
END_VAR
CASE eTestStep OF

E_BPTMTestStates.Init:
    
    TEST('BPTMErrorFullArb');
    
    // Fill the arbiter
    FOR idx := 1 TO PMPS_GVL.MAX_ASSERTIONS // this fills the arbiter
                    - fbBPTM_TestFullArb.cReqArbCapacity + 1 DO // but test just one over the allowed amount
        fbArbFullErr.AddRequest(nReqID := idx, stReqBP := testReq);
    END_FOR
    
    fbSubSysIO.AutoUpdateBP := TRUE;
    
    AssertTrue(PMPS_GVL.MAX_ASSERTIONS - fbArbFullErr.nEntryCount < fbBPTM_TestFullArb.cReqArbCapacity,
        'Arbiter is not full enough, rest of tests will be invalid'); 
    
    eTestStep := E_BPTMTestStates.Error;

E_BPTMTestStates.Error:
    
    TEST('BPTM Full Error');

    IF fbBPTM_TestFullArb.bError THEN
        
        AssertTrue(fbBPTM_TestFullArb.bError AND fbBPTM_TestFullArb.nErrId = PMPS_CODES.NoRoomInArb,
            'Incorrect error response from full arbiter.');
            
        TEST_FINISHED_NAMED('BPTM Full Error');
        
        eTestStep := E_BPTMTestStates.Retry;
        
	END_IF
    
E_BPTMTestStates.Retry:
    
    TEST('Test Retry Post Failed Final');
    
    // Clear the arbiter
    if entryToRetry THEN
        FOR idx := 1 TO PMPS_GVL.MAX_ASSERTIONS + 1 DO
            fbArbFullErr.RemoveRequest(idx);
        END_FOR
        entryToRetry := FALSE;
    END_IF
    
    // Push the retry button
    fbBPTM_TestFullArb.bRetry := TRUE;
    
    tonRetryTimeout(IN:=TRUE);
    
    IF tonRetryTimeout.Q OR fbBPTM_TestFullArb.q_xTransitionAuthorized THEN
        AssertTrue(fbBPTM_TestFullArb.q_xTransitionAuthorized, 'Transition should have been authorized by now');
        AssertTrue(fbArbFullErr.CheckRequest(nTransitionID), 'Transition ID is missing from arbiter while transition is authorized');
        AssertTrue(fbArbFullErr.CheckRequest(nReqID), 'Final ID is missing from arbiter while transition is authorized');
        
        TEST_FINISHED_NAMED('Test Retry Post Failed Final');
        
        eTestStep := E_BPTMTestStates.CleaningUp;
	END_IF

E_BPTMTestStates.CleaningUp:
    TEST_FINISHED_NAMED('BPTMErrorFullArb');    
    
END_CASE

fbBPTM_TestFullArb(
    fbArbiter := fbArbFullErr,
    i_TransitionAssertionID := nTransitionID,
    i_stTransitionAssertion := stTransitionAssertion,
    
    i_nRequestedAssertionID := nReqID,
    i_stRequestedAssertion := stReqAssertion,
    
    stCurrentBeamParameters := fbSubSysIO.q_stSimulatedBPReadback,
);

fbSubSysIO(LA := fbArbFullErr, FFO := ffo);
END_METHOD

END_FUNCTION_BLOCK

// TestComponents/FB_DiffBP_Test
{attribute 'call_after_init'}
FUNCTION_BLOCK FB_DiffBP_Test EXTENDS TcUnit.FB_TestSuite
VAR_INPUT
END_VAR
VAR_OUTPUT
END_VAR
VAR

END_VAR


BPDiff();

//Verify BP comparison remains logical.
METHOD BPDiff
VAR_INPUT
END_VAR
VAR
    BP1    :    ST_BeamParams;
    BP2    :    ST_BeamParams;
END_VAR
TEST('BPDiffCheck');

BP2.nTran := 10; 
    
AssertTrue(
    F_DifferentBeamParams(BP1, BP2),
    'DifferentBP eval is broken (True)'); 

BP1.nTran := BP2.nTran;   
    
AssertFalse(
    F_DifferentBeamParams(BP2, BP1),
    'DifferentBP eval is broken (False)');

TEST_FINISHED();
END_METHOD

END_FUNCTION_BLOCK

// TestComponents/FB_evRangeCalculator_Test
{attribute 'call_after_init'}
FUNCTION_BLOCK FB_evRangeCalculator_Test EXTENDS FB_TestSuite
VAR_INPUT
END_VAR
VAR_OUTPUT
END_VAR
VAR
END_VAR
VAR CONSTANT
    RandomBoundary : INT := 2;
END_VAR

BasicFunction();

METHOD BasicFunction
VAR_INPUT
END_VAR
VAR
    {attribute 'displaymode' := 'binary'}
    LastWord : WORD := 2#0000_0000_0000_0010;
    {attribute 'displaymode' := 'binary'}
    Result : WORD;
    {attribute 'displaymode' := 'binary'}
    TestEV : WORD;
    
    {attribute 'displaymode' := 'binary'}
    tEvW : WORD;
    tEv : REAL;
    
    
    fbStr : FB_FormatString;
    
    MiscNumber : INT;
END_VAR
VAR CONSTANT
    nLowerLimitBoundary : INT := 0;
    
    RandomBoundary : INT := 2;
    MNU : INT := 3; //RandomBoundary + 1
    MND : INT := 1; //RandomBoundary - 1
END_VAR
Test('CheckRanges');

//Lower limit equal
tEvW.nLowerLimitBoundary := TRUE;
tEv := PMPS_GVL.g_areVBoundaries[nLowerLimitBoundary];
Result := F_eVRangeCalculator(tEv, 0);
AssertTrue(
    Result = tEvW,
    'Lower limit not inclusive');
    
// Lower range flags
tEvW.nLowerLimitBoundary := TRUE;
tEv := PMPS_GVL.g_areVBoundaries[nLowerLimitBoundary] / 2;
Result := F_eVRangeCalculator(tEv, 0);
AssertTrue(
    Result = tEvW,
    'eV below lower range should come back true');
    
//Mid range
tEvW := 0;
tEvW.RandomBoundary := TRUE;
//ev result that is smack dab in the middle of a range
tEv := PMPS_GVL.g_areVBoundaries[RandomBoundary] - ((PMPS_GVL.g_areVBoundaries[RandomBoundary] - PMPS_GVL.g_areVBoundaries[MND]) / 2);
Result := F_eVRangeCalculator(tEv, 0);
AssertTrue(
    Result = tEvW,
    'In range failed, whatever you did, it broke this really bad.');

//Out of range
tEvW := 0;
tEvW.RandomBoundary := TRUE;
//Ev result that is beyond the current range (midway into the next range up)
tEv := PMPS_GVL.g_areVBoundaries[MNU] - (PMPS_GVL.g_areVBoundaries[MNU]-PMPS_GVL.g_areVBoundaries[RandomBoundary])/2;
Result := F_eVRangeCalculator(tEv, 0);
AssertFalse(
    Result = tEvW,
    'Out of range failed, whatever you did, it broke this really bad.');

TEST_FINISHED();

Test('Negative eV failsafes');
//Negative eV
AssertTrue(
    F_eVRangeCalculator(-300, 0) = 16#FFFF,
    'Working with antimatter? Negative eV should failsafe to FFFF.');    

TEST_FINISHED();

Test('Check hyst keeps');

LastWord := F_eVRangeCalculator(PMPS_GVL.g_areVBoundaries[RandomBoundary], 2#0000_0000_0000_0000);

// Last word should be 2#0000_0000_0000_0100

    Result := F_eVRangeCalculator(
        PMPS_GVL.g_areVBoundaries[RandomBoundary] + PMPS_GVL.reVHyst - PMPS_GVL.reVHyst/2,
         LastWord);
    TestEV := 0;
    TestEV.RandomBoundary := TRUE;
    TestEV.MNU := True;
 
    fbStr.arg1 := F_WORD(Result);
    fbStr.arg2 := F_WORD(TestEV);
    fbStr.sFormat := 'Moving up does not stick. Result: %b vs. Test: %b';
    fbStr();
        
AssertTrue(Result = TestEV,
    fbStr.sOut);
    
    Result := F_eVRangeCalculator(
        PMPS_GVL.g_areVBoundaries[RandomBoundary - 1] - PMPS_GVL.reVHyst + PMPS_GVL.reVHyst/2, 
        LastWord);
    TestEV := 0;
    TestEV.RandomBoundary := TRUE;
    TestEV.MND := True;
    
    fbStr.arg1 := F_WORD(Result);
    fbStr.arg2 := F_WORD(TestEV);
    fbStr.sFormat := 'Moving down does not stick. Result: %b vs. Test: %b';
    fbStr();
    
AssertTrue(Result = TestEV,
    fbStr.sOut);

TEST_FINISHED();

Test('Check hyst drops');

    Result := F_eVRangeCalculator(
        PMPS_GVL.g_areVBoundaries[MND] - PMPS_GVL.reVHyst*1.1, 
        LastWord);
    TestEV := 0;
    TestEV.MND := TRUE;
    
    fbStr.arg1 := F_WORD(Result);
    fbStr.arg2 := F_WORD(TestEV);
    fbStr.sFormat := 'Moving down does not drop. Result: %b vs. Test: %b';
    fbStr();
    
AssertTrue(Result = TestEV,
    fbStr.sOut);

    Result := F_eVRangeCalculator(
        PMPS_GVL.g_areVBoundaries[RandomBoundary] + PMPS_GVL.reVHyst*1.1, 
        LastWord);
    TestEV := 0;
    TestEV.MNU := TRUE;
    
    fbStr.arg1 := F_WORD(Result);
    fbStr.arg2 := F_WORD(TestEV);
    fbStr.sFormat := 'Moving up does not drop. Result: %b vs. Test: %b';
    fbStr();
    
AssertTrue(Result = TestEV,
    fbStr.sOut);

TEST_FINISHED();
END_METHOD

END_FUNCTION_BLOCK

// TestComponents/FB_eVWithinSpec_Test
{attribute 'call_after_init'}
FUNCTION_BLOCK FB_eVWithinSpec_Test EXTENDS TcUnit.FB_TestSuite
VAR_INPUT
END_VAR
VAR_OUTPUT
END_VAR
VAR
END_VAR

evWithinRangeChecks();

METHOD evWithinRangeChecks
VAR_INPUT
END_VAR
VAR

END_VAR
TEST('evWithinRangeChecks');
    
//Upper limit equal
AssertTrue(
    F_eVWithinSpec(300, 2#0000_0000_0000_0010),
    'Upper limit not inclusive');
//Lower limit equal
AssertTrue(
    F_eVWithinSpec(300, 2#0000_0000_0000_0100),
    'Lower limit not inclusive');
//Out of range
AssertFalse(
    F_eVWithinSpec(300.1, 2#0000_0000_0000_0010),
    'Out of range failed, whatever you did, it broke this really bad.');
//Negative eV
AssertFalse(
    F_eVWithinSpec(-300, 16#FFFF),
    'Working with antimatter? Negative eV should not be acceptable.');
//Upper unallocated range
AssertFalse(
    F_eVWithinSpec(1701, 2#1000_0000_0000_0000),
    'eV range should not evaluate past 1.7keV');
    
TEST_FINISHED();
END_METHOD

END_FUNCTION_BLOCK

// TestComponents/FB_FastFault_Test
{attribute 'call_after_init'}
FUNCTION_BLOCK FB_FastFault_Test EXTENDS TcUnit.FB_TestSuite
VAR_INPUT
END_VAR
VAR_OUTPUT
END_VAR
VAR

END_VAR
VAR CONSTANT
    OvrdTime : TIME := T#2s;
END_VAR

FFCombinedFunctionality();
FFRegistration();
FFOvrdAndNextFault();

METHOD FFCombinedFunctionality
VAR_INPUT
END_VAR
VAR_INST
    fbFF    :    FB_FastFault;
    fbFFO    :    FB_HardwareFFOutput;
    
END_VAR
TEST('FFCombinedFunctionality');

//Clear initial faults
fbFFO.i_xReset:=TRUE; //Reset requested at start of cycle

fbFF(io_fbFFHWO := fbFFO, //FF reset somehwere in code
    i_xOK := TRUE,
    i_xReset := TRUE);

fbFFO.EvaluateOutput(); //FFO eval called at end of cycle
    
AssertTrue(fbFFO.q_xFastFaultOut,
    'Fast fault did not clear');


//Induce fault with FF

fbFFO(i_xReset := FALSE); //Reset released at start of cycle

fbFF(io_fbFFHWO := fbFFO, //FF faulted
    i_xOK := FALSE); //Reset is still set true from last call.
    
fbFFO.EvaluateOutput(); //FFO eval called at end of cycle

AssertFalse(fbFFO.q_xFastFaultOut,
    'Fast fault did not trip the beam');
    
    
//FFO remains faulted until local (FF) and FFO receieve fresh reset request, and faults
//are actually cleared

//Attempt to clear FFO fails because FF still faulted
fbFFO.i_xReset := TRUE; //Reset requested

fbFF(io_fbFFHWO := fbFFO, //FF faulted
    i_xOK := FALSE,
    i_xReset := FALSE);
    
fbFFO.EvaluateOutput(); //FFO eval called at end of cycle

AssertFalse(fbFFO.q_xFastFaultOut,
    'Fast fault output cleared while fault remains, very bad');
    
//Attempt to clear FF while fault remains fails
fbFFO.EvaluateOutput(i_xReset := FALSE);

fbFFO.i_xReset := TRUE; //Reset requested

fbFF(io_fbFFHWO := fbFFO, //FF faulted
    i_xOK := FALSE,
    i_xReset := TRUE); //This reset should fail.
    
fbFFO.EvaluateOutput(); //FFO eval called at end of cycle

AssertFalse(fbFFO.q_xFastFaultOut,
    'Fast fault cleared while fault remains, very bad');
    
TEST_FINISHED();
END_METHOD

METHOD FFOvrdAndNextFault
VAR_INPUT
END_VAR
VAR_INST
    fbFF    :    FB_FastFault :=(
        i_xAutoReset := TRUE);
    fbFFO    :    FB_HardwareFFOutput := (
        bAutoReset := TRUE);
    rFF : REFERENCE TO ST_FF;
    
    FirstPass : BOOL := TRUE;
    OvrdActvTstDone : BOOL := FALSE;
    
    TestsDone : BOOL := FALSE;
END_VAR
TEST('FFVetoAndNextFault');

// I noticed something weird going on with the PEWatcher on the L line. It was faulted, and the fast fault
// was not tripping off beam. It had been previously overridden so I was wondering why it wasn't causing a trip.

IF FirstPass THEN

    fbFF(io_fbFFHWO := fbFFO, //FF reset somehwere in code
        i_xOK := TRUE);
    
    fbFFO.ExecuteNoLog(); //FFO eval called at end of cycle
        
    AssertTrue(fbFFO.q_xFastFaultOut,
        'Fast fault did not clear');
    
    
    //Induce fault with FF
    
    fbFF(io_fbFFHWO := fbFFO, //FF faulted
        i_xOK := FALSE); 
        
    fbFFO.ExecuteNoLog(); //FFO eval called at end of cycle
    
    AssertFalse(fbFFO.q_xFastFaultOut,
        'Fast fault did not trip the beam');


    rFF REF= fbFFO.astFF[fbFF.RegistrationIdx];

    
    // Overrides set from EPICS
    WRITE_PROTECTED_TIME(ADR(rFF.Ovrd.Duration), OvrdTime);
    WRITE_PROTECTED_BOOL(ADR(rFF.Ovrd.Activate), TRUE);
    
    
    FirstPass := FALSE;
    
END_IF

// On every cycle:
fbFF(io_fbFFHWO := fbFFO, //FF faulted
    i_xOK := FALSE); 
    
fbFFO.ExecuteNoLog(); //FFO eval called at end of cycle


IF rFF.Ovrd.Active AND rFF.BeamPermitted THEN

    AssertTrue(fbFFO.q_xFastFaultOut,
        'Fast fault should be overridden so FFO should be true');
    
    OvrdActvTstDone := TRUE;
END_IF

IF OvrdActvTstDone and NOT rFF.Ovrd.Active and not rff.BeamPermitted THEN
    
    AssertFalse(fbFFO.q_xFastFaultOut,
        'Fast fault override expired so beam should be off.');
   // AssertFalse(rFF.BeamPermitted, 'Beam should not be permitted now');
    
    TestsDone := TRUE;
END_IF


IF TestsDone THEN    
    TEST_FINISHED_NAMED('FFVetoAndNextFault');
END_IF
END_METHOD

METHOD FFRegistration
VAR_INPUT
END_VAR
VAR_INST
    fbFF    :    FB_FastFault;
    fbFFO    :    FB_HardwareFFOutput;
    astFF : ARRAY[0..10] OF ST_FF;
END_VAR
TEST('FFRegistration');

fbFF(io_fbFFHWO := fbFFO);

AssertEquals_STRING(fbFF.sPath, fbFFO.astFF[fbFF.RegistrationIdx].Info.sPath,
    'FF registration with FFO did not succeed');

TEST_FINISHED();
END_METHOD

END_FUNCTION_BLOCK

// TestComponents/FB_PhotonEnergyWatcher_Test
{attribute 'call_after_init'}
FUNCTION_BLOCK FB_PhotonEnergyWatcher_Test EXTENDS TcUnit.FB_TestSuite
VAR_INPUT
END_VAR
VAR_OUTPUT
END_VAR
VAR

END_VAR

PEWatcherBasicFunction();

METHOD PEWatcherBasicFunction
VAR_INPUT
END_VAR
VAR_INST
    fbPEW    :    FB_PhotonEnergyWatcher;
    fbFFO    :    FB_HardwareFFOutput;
    q_Output    :    BOOL;
    
    stCurBeamParams    :    ST_BeamParams;
    stMachineTargetBeamParams    :    ST_BeamParams;
    stReqBeamParams    :    ST_BeamParams;
END_VAR
TEST('PEWatcherBasicFunction');

//Clear FFO fault to start
fbFFO(i_xReset:=TRUE);

//All eV OK
stCurBeamParams.neVRange := F_eVRangeCalculator(800, 0);
    
stMachineTargetBeamParams.neVRange := 2#0000_0000_1000_0000;

stReqBeamParams.neVRange := 2#1111_1111_1111_1111;    

fbFFO(i_xReset:=FALSE); //Reset request released
    
fbPEW(i_stCurrentBeamParams := stCurBeamParams,
    i_stMachineTargetBeamParams := stMachineTargetBeamParams,
    i_stRequestedBeamParams := stReqBeamParams,
    io_fbFFHWO := fbFFO,
    i_xReset := TRUE); //Clear local FF within PEW
    
fbFFO.EvaluateOutput(q_xFastFaultOut=>q_Output); //This simulates a completed PLC cycle
//Evaluate output should be called once at the end of a PLC cycle.

AssertTrue(q_Output,
    'Beam within limits, FFO should be true');
    
    
//Req eV moved out of range
stCurBeamParams.neVRange := F_eVRangeCalculator(800, 0);
    
stMachineTargetBeamParams.neVRange := F_eVRangeCalculator(800, 0);

stReqBeamParams.neVRange := 2#0000_1111_0011_1111;

fbPEW.i_xReset := FALSE; //release local FF reset req    
fbPEW(i_stCurrentBeamParams := stCurBeamParams,
    i_stMachineTargetBeamParams := stMachineTargetBeamParams,
    i_stRequestedBeamParams := stReqBeamParams,
    io_fbFFHWO := fbFFO);
    
fbFFO.EvaluateOutput(q_xFastFaultOut=>q_Output);

AssertFalse(q_Output,
    'Limits moved beyond current and target beam, should produce a fault.');

//Beam and target eV moved back within permitted ranges, reset clears fault
stCurBeamParams.neVRange := F_eVRangeCalculator( 300, 0);
    
stMachineTargetBeamParams.neVRange := F_eVRangeCalculator(300, 0);

stReqBeamParams.neVRange := 2#0000_1111_0011_1111;

fbFFO(i_xReset:=TRUE); //New reset request

fbPEW.i_xReset := TRUE; //New reset request

fbPEW(i_stCurrentBeamParams := stCurBeamParams, //Beam params are now within spec
    i_stMachineTargetBeamParams := stMachineTargetBeamParams,
    i_stRequestedBeamParams := stReqBeamParams,
    io_fbFFHWO := fbFFO);
    
fbFFO.EvaluateOutput(q_xFastFaultOut=>q_Output);

AssertTrue(q_Output,
    'Beam within limits after reset, FFO should be true');
    
//At this point, the fast fault would be cleared

//Current beam eV moved out of range
stCurBeamParams.neVRange := F_eVRangeCalculator(800, 0); //Moved out of range
    
stMachineTargetBeamParams.neVRange := F_eVRangeCalculator(300, 0); //Still within range

stReqBeamParams.neVRange := 2#0000_1111_0011_1111;

fbPEW(i_stCurrentBeamParams := stCurBeamParams,
    i_stMachineTargetBeamParams := stMachineTargetBeamParams,
    i_stRequestedBeamParams := stReqBeamParams,
    io_fbFFHWO := fbFFO);
    
fbFFO.EvaluateOutput(q_xFastFaultOut=>q_Output);

AssertFalse(q_Output,
    'Current beam moved beyond set limits, should produce a fault');

//Target beam eV moved out of range
fbFFO(i_xReset:=FALSE); //Reset released
fbFFO(i_xReset:=TRUE); //New reset request comes in at the top of a cycle, but will be overridden

stCurBeamParams.neVRange := F_eVRangeCalculator(300, 0); //Now within range
    
stMachineTargetBeamParams.neVRange := F_eVRangeCalculator(800, 0); //Moved out of range

stReqBeamParams.neVRange := 2#0000_1111_0011_1111;

fbPEW.i_xReset := TRUE; //Attempt to reset local FF will fail
fbPEW(i_stCurrentBeamParams := stCurBeamParams,
    i_stMachineTargetBeamParams := stMachineTargetBeamParams,
    i_stRequestedBeamParams := stReqBeamParams,
    io_fbFFHWO := fbFFO);
    
fbFFO.EvaluateOutput(q_xFastFaultOut=>q_Output);

AssertFalse(q_Output,
    'Target beam moved beyond set limits, should produce a fault');
    
TEST_FINISHED();
END_METHOD

END_FUNCTION_BLOCK

// TestComponents/FB_SafeBPCompare_Test
{attribute 'call_after_init'}
FUNCTION_BLOCK FB_SafeBPCompare_Test EXTENDS TcUnit.FB_TestSuite
VAR_INPUT
END_VAR
VAR_OUTPUT
END_VAR
VAR

END_VAR

BeamOffIsSafe();
BPComparisonCheck();

//Verify beam off is considered safe.
METHOD BeamOffIsSafe
VAR_INPUT
END_VAR
VAR
    stBeamOn_MoreConservative    :    ST_BeamParams;
    stBeamOff_LessConservative    :    ST_BeamParams;
END_VAR
stBeamOn_MoreConservative  := F_SetBeamParams(
    50, //50% attenuation is more conservative than 0
    10,
    16#FFFF,
    120, //rate
    PMPS_GVL.DUMMY_AUX_ATT_ARRAY);

stBeamOff_LessConservative:= F_SetBeamParams(
    0, //0% attenuation, less conservative, without 0-rate this beam parameter set would be less safe than above
    10,
    16#FFFF,
    0, //rate, hence, more conservative
    PMPS_GVL.DUMMY_AUX_ATT_ARRAY); //0 beam rate means this bps is actually safer than BeamOn

TEST('BeamOffIsSafe');
    
AssertTrue(
    F_SafeBPCompare(stBeamOff_LessConservative, stBeamOn_MoreConservative),
    'SafeBPCompare does not think beam rate = 0 is safer than anything else.'); 
TEST_FINISHED();
END_METHOD

//Verify BP comparison remains logical.
METHOD BPComparisonCheck
VAR_INPUT
END_VAR
VAR
    stSafer    :    ST_BeamParams;
    stNotSoSafe    :    ST_BeamParams;
    idx : UINT;
END_VAR


TEST('BPComparisonTran');
//Attenuation
stSafer := F_SetBeamParams(
    0, //
    10,
    16#FFFF,
    1,
    PMPS_GVL.DUMMY_AUX_ATT_ARRAY);

stNotSoSafe := F_SetBeamParams(
    1, //
    10,
    16#FFFF,
    1,
    PMPS_GVL.DUMMY_AUX_ATT_ARRAY); 
    
AssertTrue(
    F_SafeBPCompare(stSafer, stNotSoSafe),
    'Attenuation eval is broken (True)'); 

AssertFalse(
    F_SafeBPCompare(stNotSoSafe, stSafer),
    'Attenuation eval is broken (False)');

TEST_FINISHED();
    
//Attenuator array    
TEST('BPComparisonTranArray');

stNotSoSafe := F_SetBeamParams(
    0, //
    10,
    16#FFFF,
    1,
    PMPS_GVL.DUMMY_AUX_ATT_ARRAY); 

FOR idx:=1 TO PMPS_GVL.AUX_ATTENUATORS DO
    stSafer.astAttenuators[idx].nTran := 30;
    stNotSoSafe.astAttenuators[idx].nTran := 50;
    
    AssertTrue(
    F_SafeBPCompare(stSafer, stNotSoSafe),
    'Attenuation array eval is broken (True)'); 

    AssertFalse(
    F_SafeBPCompare(stNotSoSafe, stSafer),
    'Attenuation array eval is broken (False)');
    
    IF NOT F_SafeBPCompare(stSafer, stNotSoSafe) or F_SafeBPCompare(stNotSoSafe, stSafer) THEN
        EXIT; // Exit this loop on the first failure.
	END_IF
    
    stSafer.astAttenuators[idx].nTran := 0;
    stNotSoSafe.astAttenuators[idx].nTran := 0;
    
END_FOR

TEST_FINISHED();

stSafer.astAttenuators[idx].nTran := 0;
stNotSoSafe.astAttenuators[idx].nTran := 0;

//Aperture array
TEST('BPComparisonApertureArray');

FOR idx:=1 TO PMPS_GVL.MAX_APERTURES DO
    // Height
    stSafer.astApertures[idx].Height := 30; // narrower is safer
    stNotSoSafe.astApertures[idx].Height := 50;
    
    AssertTrue(
    F_SafeBPCompare(stSafer, stNotSoSafe),
    'Aperture array eval is broken on height (True)'); 

    AssertFalse(
    F_SafeBPCompare(stNotSoSafe, stSafer),
    'Aperture array eval is broken on height (False)');
    
    IF NOT F_SafeBPCompare(stSafer, stNotSoSafe) or F_SafeBPCompare(stNotSoSafe, stSafer) THEN
        EXIT; // Exit this loop on the first failure.
	END_IF
    
    stSafer.astApertures[idx].Height := 0;
    stNotSoSafe.astApertures[idx].Height := 0;
    
    // Width
    stSafer.astApertures[idx].Width := 30; // narrower is safer
    stNotSoSafe.astApertures[idx].Width := 50;
    
    AssertTrue(
    F_SafeBPCompare(stSafer, stNotSoSafe),
    'Aperture array eval is broken on width (True)'); 

    AssertFalse(
    F_SafeBPCompare(stNotSoSafe, stSafer),
    'Aperture array eval is broken on width (False)');
    
    IF NOT F_SafeBPCompare(stSafer, stNotSoSafe) or F_SafeBPCompare(stNotSoSafe, stSafer) THEN
        EXIT; // Exit this loop on the first failure.
	END_IF
    
    stSafer.astApertures[idx].Width := 0;
    stNotSoSafe.astApertures[idx].Width := 0;
    
    
END_FOR

TEST_FINISHED();
    
//Rate
TEST('BPComparisonRate');
stSafer := F_SetBeamParams(
    0,
    10,
    16#FFFF,
    1,
    PMPS_GVL.DUMMY_AUX_ATT_ARRAY); //

stNotSoSafe := F_SetBeamParams(
    0,
    10,
    16#FFFF,
    10,
    PMPS_GVL.DUMMY_AUX_ATT_ARRAY); //
    
AssertTrue(
    F_SafeBPCompare(stSafer, stNotSoSafe),
    'Rate eval is broken (True)'); 

AssertFalse(
    F_SafeBPCompare(stNotSoSafe, stSafer),
    'Rate eval is broken (False)');
TEST_FINISHED();
    
//Pulse energy
TEST('BPComparisonPulseEnergy');
stSafer := F_SetBeamParams(
    0, 
    1, //
    16#FFFF,
    1,
    PMPS_GVL.DUMMY_AUX_ATT_ARRAY);

stNotSoSafe := F_SetBeamParams(
    0, 
    10, //
    16#FFFF,
    1,
    PMPS_GVL.DUMMY_AUX_ATT_ARRAY); 
    
AssertTrue(
    F_SafeBPCompare(stSafer, stNotSoSafe),
    'Pulse energy eval is broken (True)'); 

AssertFalse(
    F_SafeBPCompare(stNotSoSafe, stSafer),
    'Pulse energy eval is broken (False)');    
TEST_FINISHED();
    
//Photon energy
//More extensive tests elsewhere
TEST('BPComparisonPhotonEnergy');
stSafer := F_SetBeamParams(
    0, 
    1, 
    2#0000_0000_0000_0010,
    1,
    PMPS_GVL.DUMMY_AUX_ATT_ARRAY);

stNotSoSafe := F_SetBeamParams(
    0, 
    1, 
    2#0000_0000_0000_0110,
    1,
    PMPS_GVL.DUMMY_AUX_ATT_ARRAY);
    
AssertTrue(
    F_SafeBPCompare(stSafer, stNotSoSafe),
    'Photon energy eval is broken (True)'); 

AssertFalse(
    F_SafeBPCompare(stNotSoSafe, stSafer),
    'Photon energy eval is broken (False)');    
TEST_FINISHED();
END_METHOD

END_FUNCTION_BLOCK

// TestComponents/FB_SubsysToArb_Test
{attribute 'call_after_init'}
FUNCTION_BLOCK FB_SubsysToArb_Test EXTENDS TcUnit.FB_TestSuite
VAR_INPUT
END_VAR
VAR_OUTPUT
END_VAR
VAR
END_VAR

BasicFunction();

METHOD BasicFunction
VAR_INPUT
END_VAR
VAR   
    nId    :    DWORD := 1;
    stReq    :    ST_BeamParams := (nTran:=12);
END_VAR
VAR_INST
    fbArbiter    :    FB_Arbiter(1);
    
    fbSubSysToArb : FB_SubSysToArbiter_IO; // Subsystem interface with beamline arbiter PLC
    pBPC : POINTER TO ST_BeamParams_IO;
    
    ioCurrentBP : ST_BeamParams_IO; 
    
    FFO : FB_HardwareFFOutput; // Dummy FFO not important for these tests
    
END_VAR
VAR CONSTANT
    SysID : DWORD := 42;
END_VAR
// This simulates a synchronous cycle between the subsystem and arbiter PLC cycles. Ie. phase is locked, and cycle time is the same. This is not always the case, so these tests should be 
// trusted with a grain of salt.

TEST('Add to arbiter');

IF NOT fbArbiter.CheckRequestInPool(nID) THEN
    AssertTrue(fbArbiter.AddRequest(nId, stReq), 'Arbiter returned false from AddRequest'); // some device asking its local arbiter for some beam parameters
END_IF  
   
TEST_FINISHED();   

///////////////////////////////////////
//Sub system cycle
fbSubSysToArb(Arbiter := fbArbiter, fbFFHWO := FFO);
//END of sub system cycle
///////////////////////////////////////


TEST('Initial Elevation');
AssertTrue(fbSubSysToArb.nRequestCohort = fbSubSysToArb.q_stRequestedBP.nCohortInt, 'ReqCohort and qBP Cohort do not match');
AssertFalse(fbArbiter.xActiveInArbitration, 'Arbiter indicates it is included in arbitration prematurely');
AssertTrue(fbSubSysToArb.nRequestCohort = 1, 'Cohort index should move to 1 with first request');
TEST_FINISHED_NAMED('Initial Elevation');
    
//Ethercat transfer simulation
// Transfer of requested BP to arbiter PLC
// pBPR := ADR(fbArbToSubSys.i_RequestedBP);
// pBPR^ := fbSubSysToArb.q_stRequestedBP;

ioCurrentBP := fbSubSysToArb.q_stRequestedBP;
// NOTE: Setting the returning cohort number to something less than the request cohort number
// will prevent the sub system arbiter FB from considering itself active in arbitration.
// The next set of tests verify this.
ioCurrentBP.nCohortInt := 0;

// Transfer of current BP to sub system PLC
pBPC := ADR(fbSubSysToArb.i_stCurrentBP);
pBPC^ := ioCurrentBP;

///////////////////////////////////////
//Sub system cycle
fbSubSysToArb(Arbiter := fbArbiter, fbFFHWO := FFO);
//END of sub system cycle
///////////////////////////////////////

TEST('Not yet active in arbitration');
AssertTrue(fbSubSysToArb.nActiveCohort = 0, 'Active cohort should still be zero, per ioCurrentBP.nCohortInt setting above.');
AssertFalse(fbArbiter.xActiveInArbitration, 'Arbiter indicates it is included in arbitration prematurely, checkrequest might be broken');
AssertTrue(fbSubSysToArb.nRequestCohort = 1, 'Cohort index should remain at 1 because there have been no additional requests added to the arbiter');
TEST_FINISHED_NAMED('Not yet active in arbitration');

//Ethercat transfer simulation
// Transfer of requested BP to arbiter PLC
// pBPR := ADR(fbArbToSubSys.i_RequestedBP);
// pBPR^ := fbSubSysToArb.q_stRequestedBP;

ioCurrentBP := fbSubSysToArb.q_stRequestedBP;
// NOTE: Now we simulate the FB_ArbiterToSubSys_IO updating the cohort number to the same value as the request cohort, indicating that cohort has been included
ioCurrentBP.nCohortInt := 1;

// Transfer of current BP to sub system PLC
pBPC := ADR(fbSubSysToArb.i_stCurrentBP);
pBPC^ := ioCurrentBP;

///////////////////////////////////////
//Sub system cycle
fbSubSysToArb(Arbiter := fbArbiter, fbFFHWO := FFO);
//END of sub system cycle
///////////////////////////////////////

TEST('Active in arbitration');
AssertTrue(fbSubSysToArb.nActiveCohort = fbSubSysToArb.nRequestCohort, 'Active cohort and request cohort do not match');
AssertTrue(fbArbiter.xActiveInArbitration, 'Arbiter does not indicate it is included in higher arbitration');
TEST_FINISHED_NAMED('Active in arbitration');
END_METHOD

END_FUNCTION_BLOCK

// TestComponents/FB_VetoArbiter_Test
{attribute 'call_after_init'}
FUNCTION_BLOCK FB_VetoArbiter_Test EXTENDS TcUnit.FB_TestSuite
VAR_INPUT
END_VAR
VAR_OUTPUT
END_VAR
VAR
END_VAR
VAR CONSTANT
    ArbID : DWORD := 1;
	HigherArbID : DWORD := 2;
END_VAR

VetoArbiter();

METHOD VetoArbiter

VAR_INPUT
END_VAR
VAR   
    nId    :    DWORD := 1;
	nId2 : DWORD := 10;
    stReq    :    ST_BeamParams := (nTran:=12);
	stReq2	:	ST_BeamParams := (nTran:=10);
END_VAR
VAR_INST
    fbArbiter    :    FB_Arbiter(1);
    
    fbHigherArb : FB_Arbiter(2);
	
	ArbBP : ST_BeamParams;
	
	VetoArb : FB_VetoArbiter;
	
	FFO : FB_HardwareFFOutput;
	
	fbHA : FB_DummyHA;
    
END_VAR

TEST('VetoNotIn');
fbArbiter.AddRequest(nReqID:=nId, stReqBP:=stReq);

//////////////////// Cycle    
fbHigherArb.ElevateRequest(fbHA);

VetoArb.bVeto := FALSE;
VetoArb(HigherAuthority:=fbHigherArb,
	LowerAuthority:=fbArbiter,
	FFO:=FFO);
    
//////////////////// Cycle    
fbHigherArb.ElevateRequest(fbHA);

VetoArb.bVeto := FALSE;
VetoArb(HigherAuthority:=fbHigherArb,
	LowerAuthority:=fbArbiter,
	FFO:=FFO);

AssertTrue(fbHigherArb.q_stBeamParams.nTran = stReq.nTran, 'We should see the transmission number here, veto device is not in');

TEST_FINISHED();

TEST('VetoIn');
// Veto device is in
// This should effectively remove the fbArbiter request from the higher arbiter pool

//////////////////// Cycle    
fbHigherArb.ElevateRequest(fbHA);

VetoArb.bVeto := TRUE;
VetoArb(HigherAuthority:=fbHigherArb, // Veto removed
	LowerAuthority:=fbArbiter,
	FFO:=FFO);

//////////////////// Cycle    
fbHigherArb.ElevateRequest(fbHA);

VetoArb.bVeto := TRUE;
VetoArb(HigherAuthority:=fbHigherArb, // Veto removed
	LowerAuthority:=fbArbiter,
	FFO:=FFO);
    
AssertTrue(fbHigherArb.q_stBeamParams.nTran = PMPS_GVL.cstFullBeam.nTran, 'Veto device is in, trans should be restored to 100');
AssertTrue(fbArbiter.CheckRequest(nId), 'Request should still be considered valid (1)');
AssertFalse(fbHigherArb.CheckRequest(ArbID), 'Lower arb request should be gone from the higher pool');

TEST_FINISHED();

TEST('AnotherRequest');
// Another request is added, should be approved immediately, and with no effect on the final set
fbArbiter.RequestBP(nReqID := nId2, stReqBP:=stReq2);

//////////////////// Cycle    
fbHigherArb.ElevateRequest(fbHA);

VetoArb.bVeto := TRUE;
VetoArb(HigherAuthority:=fbHigherArb, // Veto removed
	LowerAuthority:=fbArbiter,
	FFO:=FFO);
    
//////////////////// Cycle    
fbHigherArb.ElevateRequest(fbHA);

VetoArb.bVeto := TRUE;
VetoArb(HigherAuthority:=fbHigherArb, // Veto removed
	LowerAuthority:=fbArbiter,
	FFO:=FFO);

AssertTrue(ArbBP.nTran = PMPS_GVL.cstFullBeam.nTran, 'Veto device remained in, trans should still be 100');
AssertTrue(fbArbiter.CheckRequest(nId), 'Request should still be considered valid (2)');
AssertTrue(fbArbiter.CheckRequest(nId2), '2nd Request should be considered valid');

TEST_FINISHED();

TEST('RemoveVeto');
// Removal of veto device, should produce a fault
//////////////////// Cycle    
fbHigherArb.ElevateRequest(fbHA);

VetoArb.bVeto := FALSE;
VetoArb(HigherAuthority:=fbHigherArb, // Veto removed
	LowerAuthority:=fbArbiter,
	FFO:=FFO);

AssertFalse(VetoArb.ffKeepItSecretKeepItSafe.i_xOK, 'Should produce a fast fault at this point because the request is not yet back in the pool');

//////////////////// Cycle  
fbHigherArb.ElevateRequest(fbHA);

VetoArb.bVeto := FALSE;
VetoArb(HigherAuthority:=fbHigherArb, // Veto removed
	LowerAuthority:=fbArbiter,
	FFO:=FFO);

//////////////////// Cycle    
fbHigherArb.ElevateRequest(fbHA);

VetoArb.bVeto := FALSE;
VetoArb(HigherAuthority:=fbHigherArb, // Veto removed
	LowerAuthority:=fbArbiter,
	FFO:=FFO);

//////////////////// Cycle    
fbHigherArb.ElevateRequest(fbHA);

VetoArb.bVeto := FALSE;
VetoArb(HigherAuthority:=fbHigherArb, // Veto removed
	LowerAuthority:=fbArbiter,
	FFO:=FFO);    
    
AssertTrue(VetoArb.ffKeepItSecretKeepItSafe.i_xOK, 'Fault should be gone.');

TEST_FINISHED();
END_METHOD

END_FUNCTION_BLOCK

// MAIN
PROGRAM MAIN
VAR
    fbSetPERanges : PE_Ranges;    

    fbDiffBPTest    :    FB_DiffBP_Test;
    fbBPTMTest    :    FB_BPTM_Test;
    fbSafeBPCompareTest    :    FB_SafeBPCompare_Test;
    //fbevWithinSpecTest    :    FB_evWithinSpec_Test;
    //fbPEWTest    :    FB_PhotonEnergyWatcher_Test;
    fbFFTest    :    FB_FastFault_Test;
    fbArbiterTest    :    FB_Arbiter_Test;
	fbVetoArbiterTest : FB_VetoArbiter_Test;
    fbevRangeCalcTest : FB_evRangeCalculator_Test;
    fbSubSysToArbTest : FB_SubsysToArb_Test;
    fbArbToSubSysTest : FB_ArbToSubsys_Test;
END_VAR

TcUnit.RUN();

END_PROGRAM
